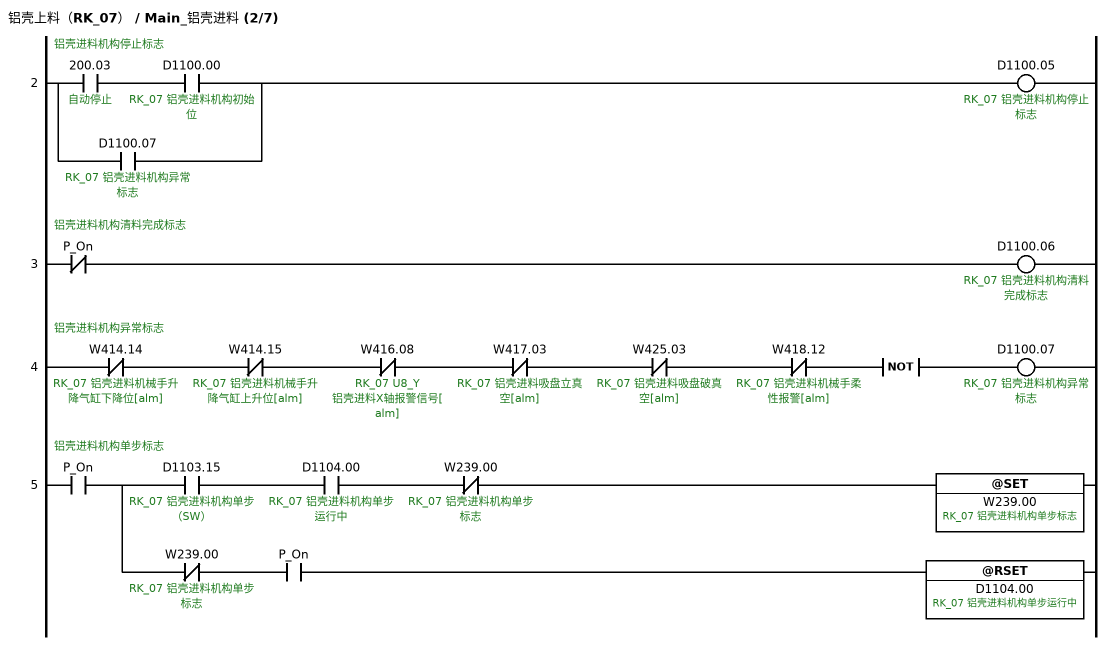
; [picture p552: 铝壳上料（RK_07） / Main_铝壳进料, rungs 2-5]
; rung 2: 铝壳进料机构停止标志
LD 200.03  ; 自动停止
AND D1100.00  ; RK_07 铝壳进料机构初始位
OR D1100.07  ; RK_07 铝壳进料机构异常标志
OUT D1100.05  ; RK_07 铝壳进料机构停止标志
; rung 3: 铝壳进料机构清料完成标志
LDNOT P_On
OUT D1100.06  ; RK_07 铝壳进料机构清料完成标志
; rung 4: 铝壳进料机构异常标志
LDNOT W414.14  ; RK_07 铝壳进料机械手升降气缸下降位[alm]
ANDNOT W414.15  ; RK_07 铝壳进料机械手升降气缸上升位[alm]
ANDNOT W416.08  ; RK_07 U8_Y 铝壳进料X轴报警信号[alm]
ANDNOT W417.03  ; RK_07 铝壳进料吸盘立真空[alm]
ANDNOT W425.03  ; RK_07 铝壳进料吸盘破真空[alm]
ANDNOT W418.12  ; RK_07 铝壳进料机械手柔性报警[alm]
NOT(520)
OUT D1100.07  ; RK_07 铝壳进料机构异常标志
; rung 5: 铝壳进料机构单步标志
LD P_On
OUT TR0
AND D1103.15  ; RK_07 铝壳进料机构单步（SW）
AND D1104.00  ; RK_07 铝壳进料机构单步运行中
ANDNOT W239.00  ; RK_07 铝壳进料机构单步标志
@SET W239.00  ; RK_07 铝壳进料机构单步标志
LD TR0
ANDNOT W239.00  ; RK_07 铝壳进料机构单步标志
AND P_On
@RSET D1104.00  ; RK_07 铝壳进料机构单步运行中

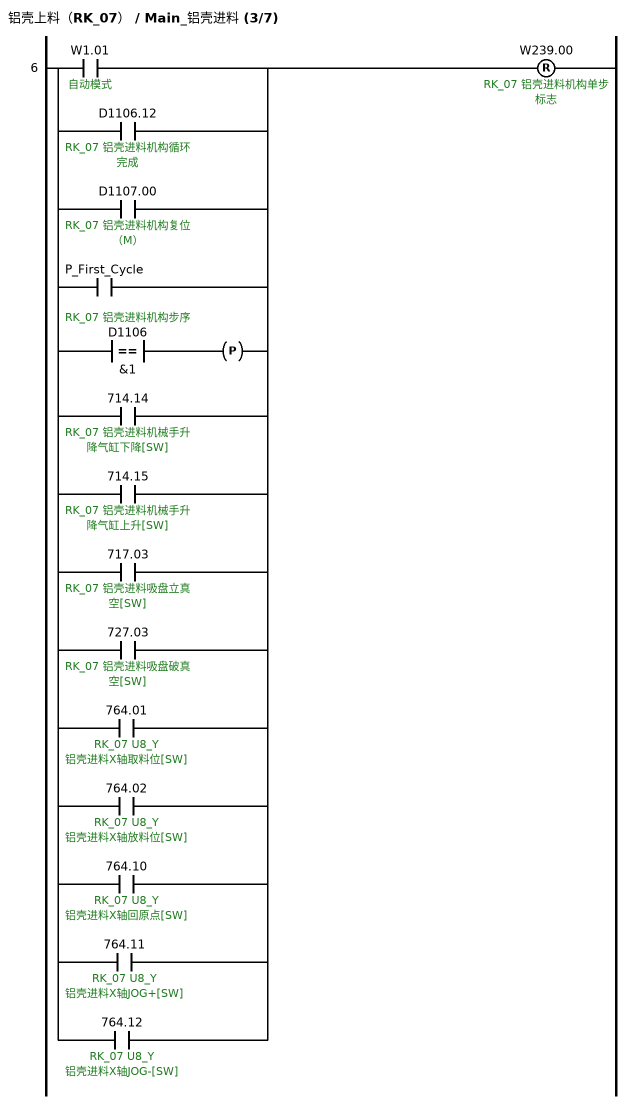
; rung 6
LD W1.01  ; 自动模式
OR D1106.12  ; RK_07 铝壳进料机构循环完成
OR D1107.00  ; RK_07 铝壳进料机构复位（M）
OR P_First_Cycle
LD=(300) D1106 &1  ; RK_07 铝壳进料机构步序
UP(521)
ORLD
OR 714.14  ; RK_07 铝壳进料机械手升降气缸下降[SW]
OR 714.15  ; RK_07 铝壳进料机械手升降气缸上升[SW]
OR 717.03  ; RK_07 铝壳进料吸盘立真空[SW]
OR 727.03  ; RK_07 铝壳进料吸盘破真空[SW]
OR 764.01  ; RK_07 U8_Y 铝壳进料X轴取料位[SW]
OR 764.02  ; RK_07 U8_Y 铝壳进料X轴放料位[SW]
OR 764.10  ; RK_07 U8_Y 铝壳进料X轴回原点[SW]
OR 764.11  ; RK_07 U8_Y 铝壳进料X轴JOG+[SW]
OR 764.12  ; RK_07 U8_Y 铝壳进料X轴JOG-[SW]
RSET W239.00  ; RK_07 铝壳进料机构单步标志

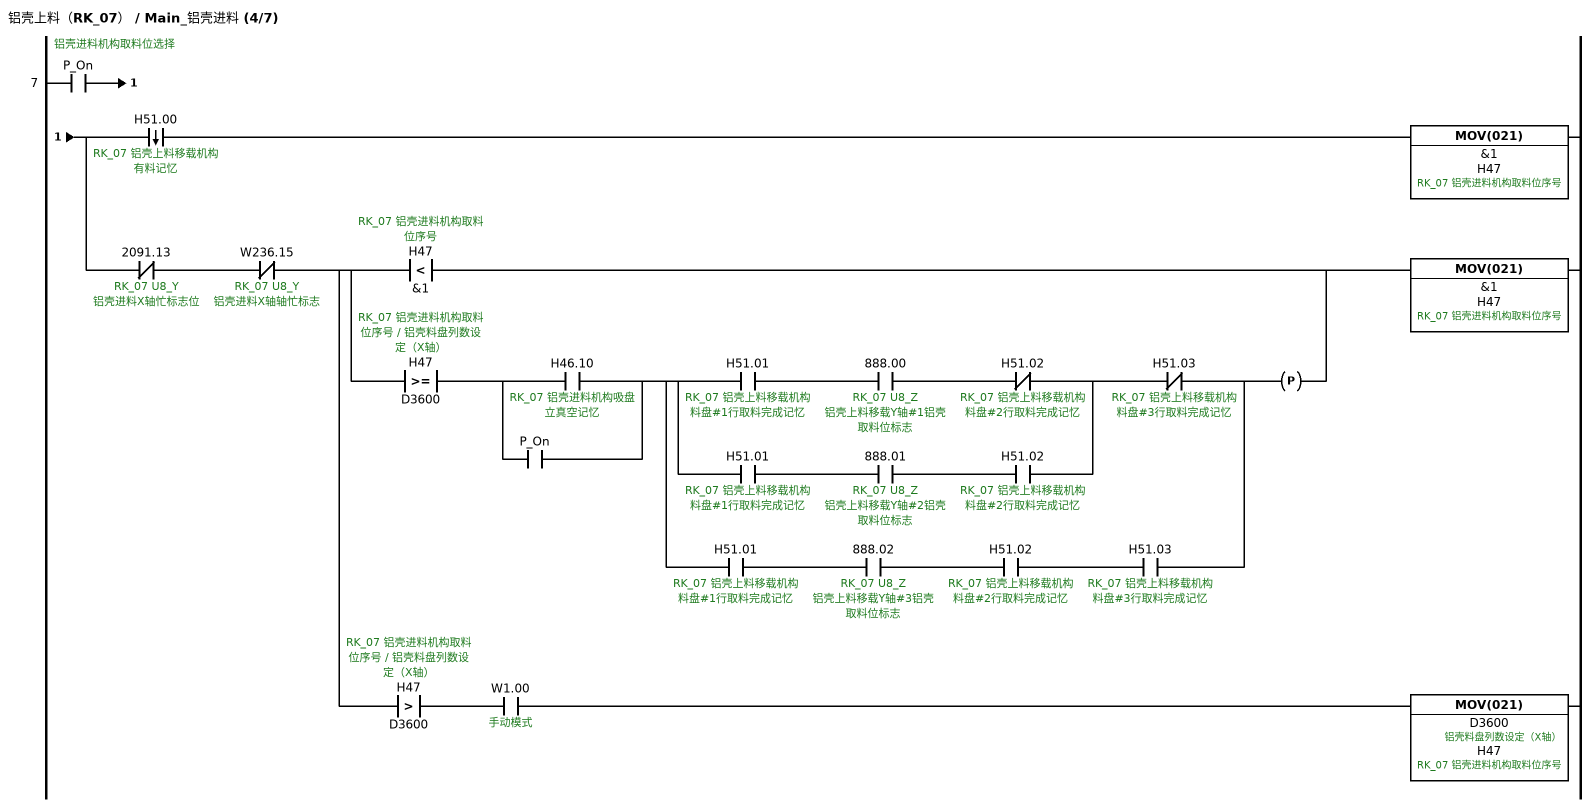
; rung 7: 铝壳进料机构取料位选择
LD P_On
OUT TR0
%AND H51.00  ; RK_07 铝壳上料移载机构有料记忆
MOV(021) &1 H47  ; RK_07 铝壳进料机构取料位序号
LD TR0
ANDNOT 2091.13  ; RK_07 U8_Y 铝壳进料X轴忙标志位
ANDNOT W236.15  ; RK_07 U8_Y 铝壳进料X轴轴忙标志
OUT TR0
LD<(310) H47 &1  ; RK_07 铝壳进料机构取料位序号
LD>=(325) H47 D3600  ; RK_07 铝壳进料机构取料位序号, 铝壳料盘列数设定（X轴）
LD H46.10  ; RK_07 铝壳进料机构吸盘立真空记忆
OR P_On
ANDLD
LD H51.01  ; RK_07 铝壳上料移载机构料盘#1行取料完成记忆
AND 888.00  ; RK_07 U8_Z 铝壳上料移载Y轴#1铝壳取料位标志
ANDNOT H51.02  ; RK_07 铝壳上料移载机构料盘#2行取料完成记忆
LD H51.01  ; RK_07 铝壳上料移载机构料盘#1行取料完成记忆
AND 888.01  ; RK_07 U8_Z 铝壳上料移载Y轴#2铝壳取料位标志
AND H51.02  ; RK_07 铝壳上料移载机构料盘#2行取料完成记忆
ORLD
ANDNOT H51.03  ; RK_07 铝壳上料移载机构料盘#3行取料完成记忆
LD H51.01  ; RK_07 铝壳上料移载机构料盘#1行取料完成记忆
AND 888.02  ; RK_07 U8_Z 铝壳上料移载Y轴#3铝壳取料位标志
AND H51.02  ; RK_07 铝壳上料移载机构料盘#2行取料完成记忆
AND H51.03  ; RK_07 铝壳上料移载机构料盘#3行取料完成记忆
ORLD
ANDLD
UP(521)
ORLD
ANDLD
MOV(021) &1 H47  ; RK_07 铝壳进料机构取料位序号
LD TR0
AND>(320) H47 D3600  ; RK_07 铝壳进料机构取料位序号, 铝壳料盘列数设定（X轴）
AND W1.00  ; 手动模式
MOV(021) D3600 H47  ; 铝壳料盘列数设定（X轴）, RK_07 铝壳进料机构取料位序号

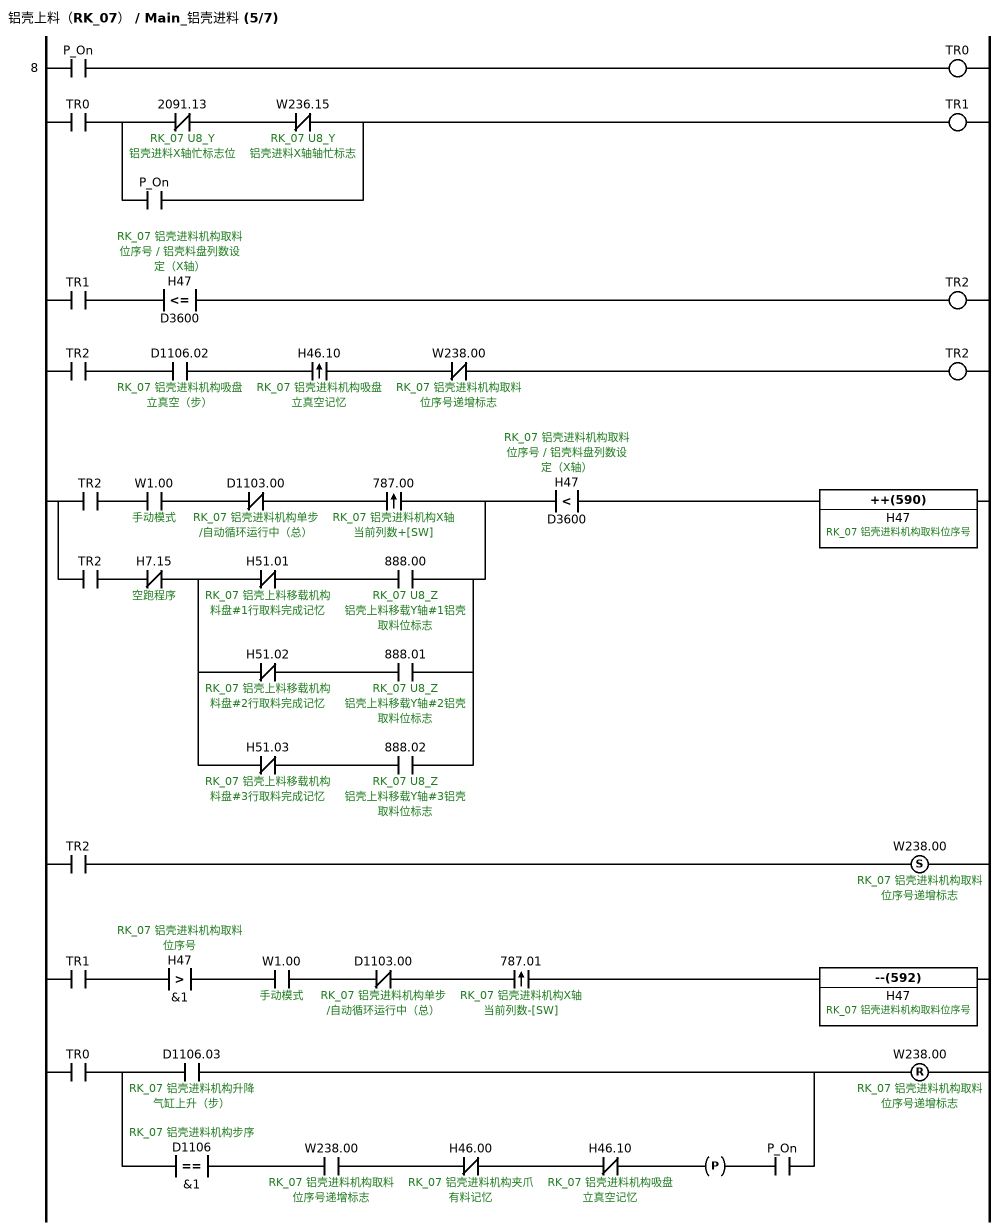
; rung 8
LD P_On
OUT TR0
LDNOT 2091.13  ; RK_07 U8_Y 铝壳进料X轴忙标志位
ANDNOT W236.15  ; RK_07 U8_Y 铝壳进料X轴轴忙标志
OR P_On
ANDLD
OUT TR1
AND<=(315) H47 D3600  ; RK_07 铝壳进料机构取料位序号, 铝壳料盘列数设定（X轴）
OUT TR2
AND W1.00  ; 手动模式
ANDNOT D1103.00  ; RK_07 铝壳进料机构单步/自动循环运行中（总）
@AND 787.00  ; RK_07 铝壳进料机构X轴当前列数+[SW]
LD TR2
AND D1106.02  ; RK_07 铝壳进料机构吸盘立真空（步）
@AND H46.10  ; RK_07 铝壳进料机构吸盘立真空记忆
ANDNOT W238.00  ; RK_07 铝壳进料机构取料位序号递增标志
OUT TR2
ANDNOT H7.15  ; 空跑程序
LDNOT H51.01  ; RK_07 铝壳上料移载机构料盘#1行取料完成记忆
AND 888.00  ; RK_07 U8_Z 铝壳上料移载Y轴#1铝壳取料位标志
LDNOT H51.02  ; RK_07 铝壳上料移载机构料盘#2行取料完成记忆
AND 888.01  ; RK_07 U8_Z 铝壳上料移载Y轴#2铝壳取料位标志
ORLD
LDNOT H51.03  ; RK_07 铝壳上料移载机构料盘#3行取料完成记忆
AND 888.02  ; RK_07 U8_Z 铝壳上料移载Y轴#3铝壳取料位标志
ORLD
ANDLD
ORLD
AND<(310) H47 D3600  ; RK_07 铝壳进料机构取料位序号, 铝壳料盘列数设定（X轴）
++(590) H47  ; RK_07 铝壳进料机构取料位序号
LD TR2
SET W238.00  ; RK_07 铝壳进料机构取料位序号递增标志
LD TR1
AND>(320) H47 &1  ; RK_07 铝壳进料机构取料位序号
AND W1.00  ; 手动模式
ANDNOT D1103.00  ; RK_07 铝壳进料机构单步/自动循环运行中（总）
@AND 787.01  ; RK_07 铝壳进料机构X轴当前列数-[SW]
--(592) H47  ; RK_07 铝壳进料机构取料位序号
LD TR0
LD D1106.03  ; RK_07 铝壳进料机构升降气缸上升（步）
LD=(300) D1106 &1  ; RK_07 铝壳进料机构步序
AND W238.00  ; RK_07 铝壳进料机构取料位序号递增标志
ANDNOT H46.00  ; RK_07 铝壳进料机构夹爪有料记忆
ANDNOT H46.10  ; RK_07 铝壳进料机构吸盘立真空记忆
UP(521)
AND P_On
ORLD
ANDLD
RSET W238.00  ; RK_07 铝壳进料机构取料位序号递增标志

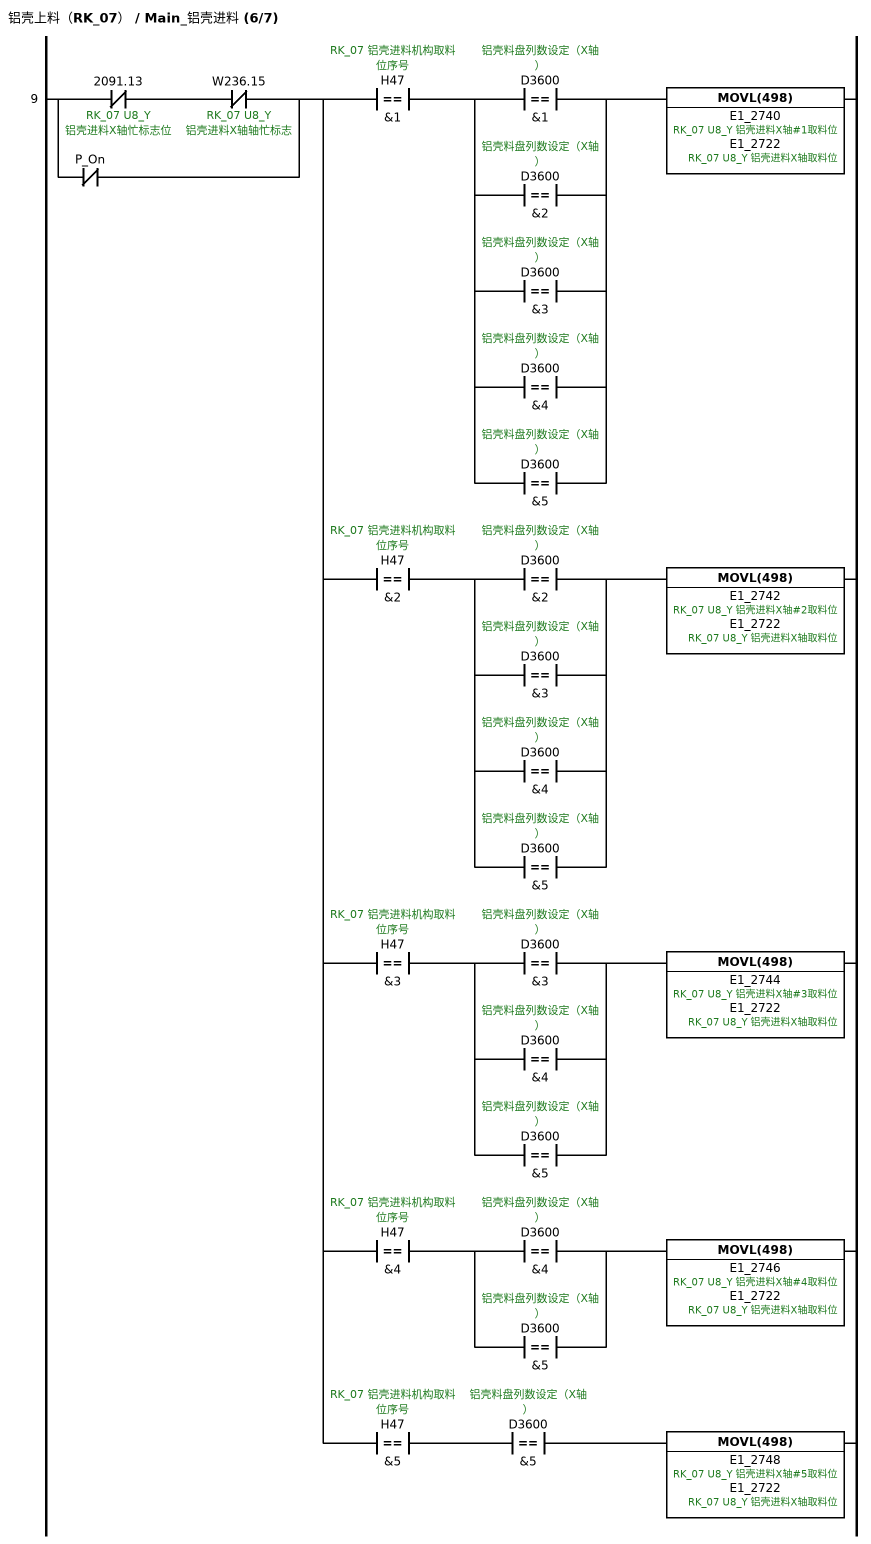
; rung 9
LDNOT 2091.13  ; RK_07 U8_Y 铝壳进料X轴忙标志位
ANDNOT W236.15  ; RK_07 U8_Y 铝壳进料X轴轴忙标志
ORNOT P_On
OUT TR0
AND=(300) H47 &1  ; RK_07 铝壳进料机构取料位序号
LD=(300) D3600 &1  ; 铝壳料盘列数设定（X轴）
OR=(300) D3600 &2  ; 铝壳料盘列数设定（X轴）
OR=(300) D3600 &3  ; 铝壳料盘列数设定（X轴）
OR=(300) D3600 &4  ; 铝壳料盘列数设定（X轴）
OR=(300) D3600 &5  ; 铝壳料盘列数设定（X轴）
ANDLD
MOVL(498) E1_2740 E1_2722  ; RK_07 U8_Y 铝壳进料X轴#1取料位, RK_07 U8_Y 铝壳进料X轴取料位
LD TR0
AND=(300) H47 &2  ; RK_07 铝壳进料机构取料位序号
LD=(300) D3600 &2  ; 铝壳料盘列数设定（X轴）
OR=(300) D3600 &3  ; 铝壳料盘列数设定（X轴）
OR=(300) D3600 &4  ; 铝壳料盘列数设定（X轴）
OR=(300) D3600 &5  ; 铝壳料盘列数设定（X轴）
ANDLD
MOVL(498) E1_2742 E1_2722  ; RK_07 U8_Y 铝壳进料X轴#2取料位, RK_07 U8_Y 铝壳进料X轴取料位
LD TR0
AND=(300) H47 &3  ; RK_07 铝壳进料机构取料位序号
LD=(300) D3600 &3  ; 铝壳料盘列数设定（X轴）
OR=(300) D3600 &4  ; 铝壳料盘列数设定（X轴）
OR=(300) D3600 &5  ; 铝壳料盘列数设定（X轴）
ANDLD
MOVL(498) E1_2744 E1_2722  ; RK_07 U8_Y 铝壳进料X轴#3取料位, RK_07 U8_Y 铝壳进料X轴取料位
LD TR0
AND=(300) H47 &4  ; RK_07 铝壳进料机构取料位序号
LD=(300) D3600 &4  ; 铝壳料盘列数设定（X轴）
OR=(300) D3600 &5  ; 铝壳料盘列数设定（X轴）
ANDLD
MOVL(498) E1_2746 E1_2722  ; RK_07 U8_Y 铝壳进料X轴#4取料位, RK_07 U8_Y 铝壳进料X轴取料位
LD TR0
AND=(300) H47 &5  ; RK_07 铝壳进料机构取料位序号
AND=(300) D3600 &5  ; 铝壳料盘列数设定（X轴）
MOVL(498) E1_2748 E1_2722  ; RK_07 U8_Y 铝壳进料X轴#5取料位, RK_07 U8_Y 铝壳进料X轴取料位

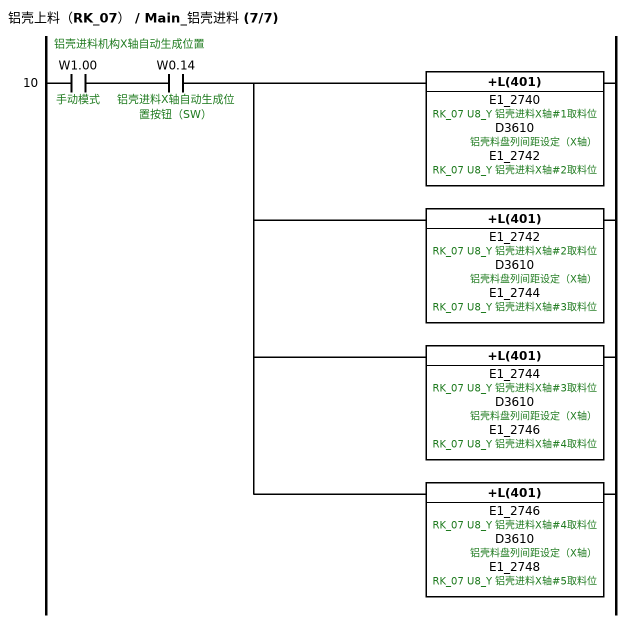
; rung 10: 铝壳进料机构X轴自动生成位置
LD W1.00  ; 手动模式
AND W0.14  ; 铝壳进料X轴自动生成位置按钮（SW）
+L(401) E1_2740 D3610 E1_2742  ; RK_07 U8_Y 铝壳进料X轴#1取料位, 铝壳料盘列间距设定（X轴）, RK_07 U8_Y 铝壳进料X轴#2取料位
+L(401) E1_2742 D3610 E1_2744  ; RK_07 U8_Y 铝壳进料X轴#2取料位, 铝壳料盘列间距设定（X轴）, RK_07 U8_Y 铝壳进料X轴#3取料位
+L(401) E1_2744 D3610 E1_2746  ; RK_07 U8_Y 铝壳进料X轴#3取料位, 铝壳料盘列间距设定（X轴）, RK_07 U8_Y 铝壳进料X轴#4取料位
+L(401) E1_2746 D3610 E1_2748  ; RK_07 U8_Y 铝壳进料X轴#4取料位, 铝壳料盘列间距设定（X轴）, RK_07 U8_Y 铝壳进料X轴#5取料位

### Section Main_铝壳上料移载

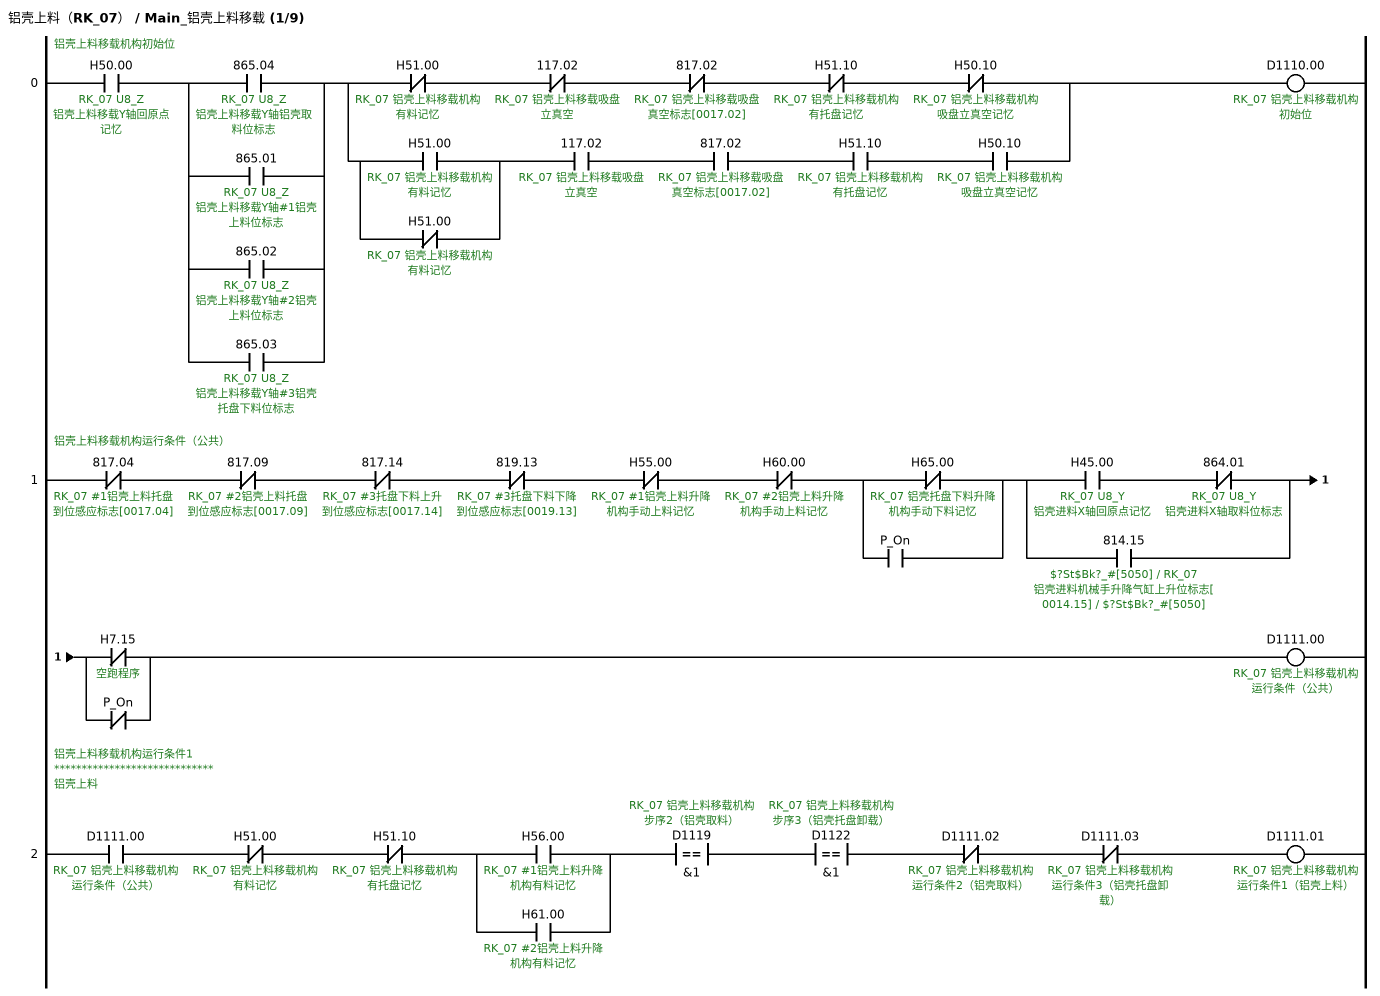
; rung 0: 铝壳上料移载机构初始位
LD H50.00  ; RK_07 U8_Z 铝壳上料移载Y轴回原点记忆
LD 865.04  ; RK_07 U8_Z 铝壳上料移载Y轴铝壳取料位标志
OR 865.01  ; RK_07 U8_Z 铝壳上料移载Y轴#1铝壳上料位标志
OR 865.02  ; RK_07 U8_Z 铝壳上料移载Y轴#2铝壳上料位标志
OR 865.03  ; RK_07 U8_Z 铝壳上料移载Y轴#3铝壳托盘下料位标志
ANDLD
LDNOT H51.00  ; RK_07 铝壳上料移载机构有料记忆
ANDNOT 117.02  ; RK_07 铝壳上料移载吸盘立真空
ANDNOT 817.02  ; RK_07 铝壳上料移载吸盘真空标志[0017.02]
ANDNOT H51.10  ; RK_07 铝壳上料移载机构有托盘记忆
ANDNOT H50.10  ; RK_07 铝壳上料移载机构吸盘立真空记忆
LD H51.00  ; RK_07 铝壳上料移载机构有料记忆
ORNOT H51.00  ; RK_07 铝壳上料移载机构有料记忆
AND 117.02  ; RK_07 铝壳上料移载吸盘立真空
AND 817.02  ; RK_07 铝壳上料移载吸盘真空标志[0017.02]
AND H51.10  ; RK_07 铝壳上料移载机构有托盘记忆
AND H50.10  ; RK_07 铝壳上料移载机构吸盘立真空记忆
ORLD
ANDLD
OUT D1110.00  ; RK_07 铝壳上料移载机构初始位
; rung 1: 铝壳上料移载机构运行条件（公共）
LDNOT 817.04  ; RK_07 #1铝壳上料托盘到位感应标志[0017.04]
ANDNOT 817.09  ; RK_07 #2铝壳上料托盘到位感应标志[0017.09]
ANDNOT 817.14  ; RK_07 #3托盘下料上升到位感应标志[0017.14]
ANDNOT 819.13  ; RK_07 #3托盘下料下降到位感应标志[0019.13]
ANDNOT H55.00  ; RK_07 #1铝壳上料升降机构手动上料记忆
ANDNOT H60.00  ; RK_07 #2铝壳上料升降机构手动上料记忆
LDNOT H65.00  ; RK_07 铝壳托盘下料升降机构手动下料记忆
OR P_On
ANDLD
LD H45.00  ; RK_07 U8_Y 铝壳进料X轴回原点记忆
ANDNOT 864.01  ; RK_07 U8_Y 铝壳进料X轴取料位标志
OR 814.15  ; $?St$Bk?_#[5050] / RK_07 铝壳进料机械手升降气缸上升位标志[0014.15] / $?St$Bk?_#[5050]
ANDLD
LDNOT H7.15  ; 空跑程序
ORNOT P_On
ANDLD
OUT D1111.00  ; RK_07 铝壳上料移载机构运行条件（公共）
; rung 2: 铝壳上料移载机构运行条件1 / ***************************** / 铝壳上料
LD D1111.00  ; RK_07 铝壳上料移载机构运行条件（公共）
ANDNOT H51.00  ; RK_07 铝壳上料移载机构有料记忆
ANDNOT H51.10  ; RK_07 铝壳上料移载机构有托盘记忆
LD H56.00  ; RK_07 #1铝壳上料升降机构有料记忆
OR H61.00  ; RK_07 #2铝壳上料升降机构有料记忆
ANDLD
AND=(300) D1119 &1  ; RK_07 铝壳上料移载机构步序2（铝壳取料）
AND=(300) D1122 &1  ; RK_07 铝壳上料移载机构步序3（铝壳托盘卸载）
ANDNOT D1111.02  ; RK_07 铝壳上料移载机构运行条件2（铝壳取料）
ANDNOT D1111.03  ; RK_07 铝壳上料移载机构运行条件3（铝壳托盘卸载）
OUT D1111.01  ; RK_07 铝壳上料移载机构运行条件1（铝壳上料）

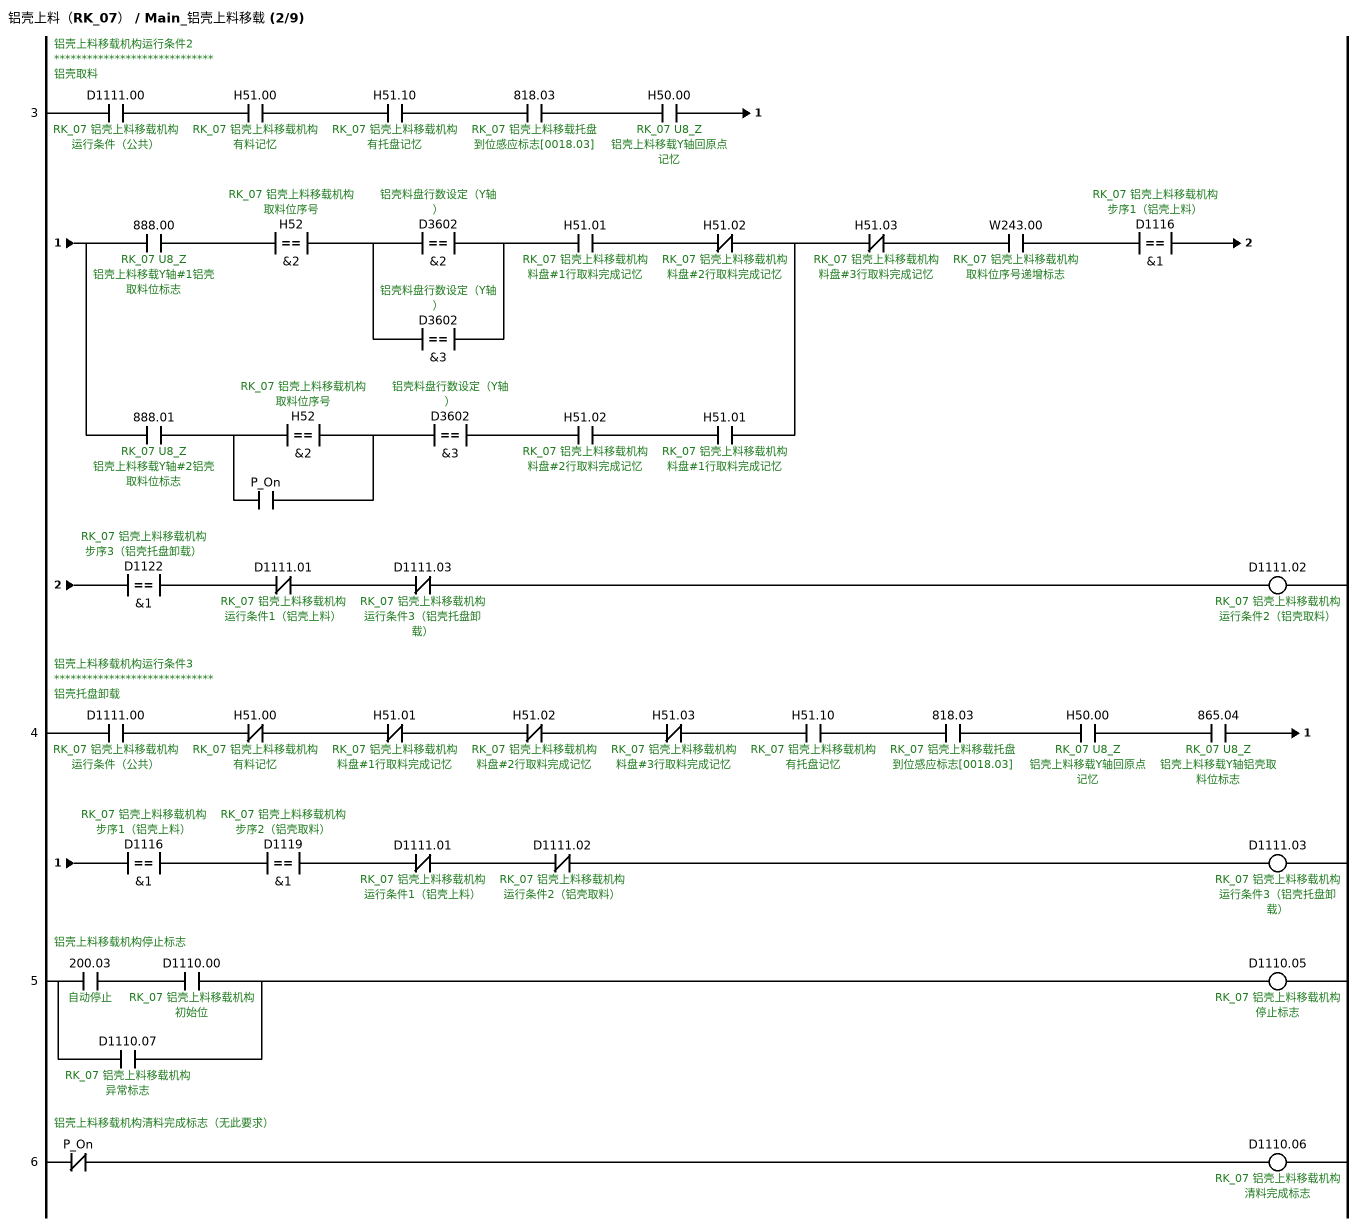
; rung 3: 铝壳上料移载机构运行条件2 / ***************************** / 铝壳取料
LD D1111.00  ; RK_07 铝壳上料移载机构运行条件（公共）
AND H51.00  ; RK_07 铝壳上料移载机构有料记忆
AND H51.10  ; RK_07 铝壳上料移载机构有托盘记忆
AND 818.03  ; RK_07 铝壳上料移载托盘到位感应标志[0018.03]
AND H50.00  ; RK_07 U8_Z 铝壳上料移载Y轴回原点记忆
LD 888.00  ; RK_07 U8_Z 铝壳上料移载Y轴#1铝壳取料位标志
AND=(300) H52 &2  ; RK_07 铝壳上料移载机构取料位序号
LD=(300) D3602 &2  ; 铝壳料盘行数设定（Y轴）
OR=(300) D3602 &3  ; 铝壳料盘行数设定（Y轴）
ANDLD
AND H51.01  ; RK_07 铝壳上料移载机构料盘#1行取料完成记忆
ANDNOT H51.02  ; RK_07 铝壳上料移载机构料盘#2行取料完成记忆
LD 888.01  ; RK_07 U8_Z 铝壳上料移载Y轴#2铝壳取料位标志
LD=(300) H52 &2  ; RK_07 铝壳上料移载机构取料位序号
OR P_On
ANDLD
AND=(300) D3602 &3  ; 铝壳料盘行数设定（Y轴）
AND H51.02  ; RK_07 铝壳上料移载机构料盘#2行取料完成记忆
AND H51.01  ; RK_07 铝壳上料移载机构料盘#1行取料完成记忆
ORLD
ANDLD
ANDNOT H51.03  ; RK_07 铝壳上料移载机构料盘#3行取料完成记忆
AND W243.00  ; RK_07 铝壳上料移载机构取料位序号递增标志
AND=(300) D1116 &1  ; RK_07 铝壳上料移载机构步序1（铝壳上料）
AND=(300) D1122 &1  ; RK_07 铝壳上料移载机构步序3（铝壳托盘卸载）
ANDNOT D1111.01  ; RK_07 铝壳上料移载机构运行条件1（铝壳上料）
ANDNOT D1111.03  ; RK_07 铝壳上料移载机构运行条件3（铝壳托盘卸载）
OUT D1111.02  ; RK_07 铝壳上料移载机构运行条件2（铝壳取料）
; rung 4: 铝壳上料移载机构运行条件3 / ***************************** / 铝壳托盘卸载
LD D1111.00  ; RK_07 铝壳上料移载机构运行条件（公共）
ANDNOT H51.00  ; RK_07 铝壳上料移载机构有料记忆
ANDNOT H51.01  ; RK_07 铝壳上料移载机构料盘#1行取料完成记忆
ANDNOT H51.02  ; RK_07 铝壳上料移载机构料盘#2行取料完成记忆
ANDNOT H51.03  ; RK_07 铝壳上料移载机构料盘#3行取料完成记忆
AND H51.10  ; RK_07 铝壳上料移载机构有托盘记忆
AND 818.03  ; RK_07 铝壳上料移载托盘到位感应标志[0018.03]
AND H50.00  ; RK_07 U8_Z 铝壳上料移载Y轴回原点记忆
AND 865.04  ; RK_07 U8_Z 铝壳上料移载Y轴铝壳取料位标志
AND=(300) D1116 &1  ; RK_07 铝壳上料移载机构步序1（铝壳上料）
AND=(300) D1119 &1  ; RK_07 铝壳上料移载机构步序2（铝壳取料）
ANDNOT D1111.01  ; RK_07 铝壳上料移载机构运行条件1（铝壳上料）
ANDNOT D1111.02  ; RK_07 铝壳上料移载机构运行条件2（铝壳取料）
OUT D1111.03  ; RK_07 铝壳上料移载机构运行条件3（铝壳托盘卸载）
; rung 5: 铝壳上料移载机构停止标志
LD 200.03  ; 自动停止
AND D1110.00  ; RK_07 铝壳上料移载机构初始位
OR D1110.07  ; RK_07 铝壳上料移载机构异常标志
OUT D1110.05  ; RK_07 铝壳上料移载机构停止标志
; rung 6: 铝壳上料移载机构清料完成标志（无此要求）
LDNOT P_On
OUT D1110.06  ; RK_07 铝壳上料移载机构清料完成标志

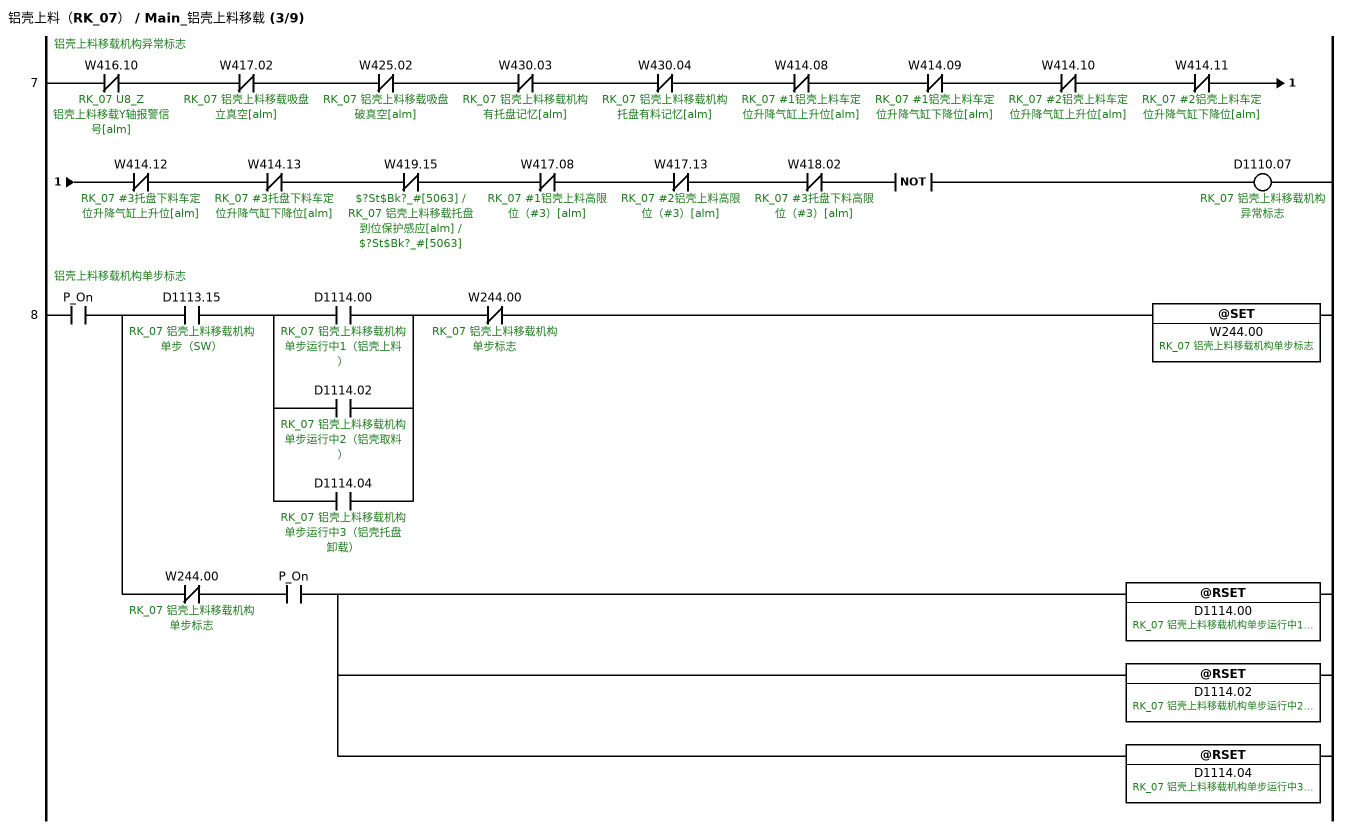
; rung 7: 铝壳上料移载机构异常标志
LDNOT W416.10  ; RK_07 U8_Z 铝壳上料移载Y轴报警信号[alm]
ANDNOT W417.02  ; RK_07 铝壳上料移载吸盘立真空[alm]
ANDNOT W425.02  ; RK_07 铝壳上料移载吸盘破真空[alm]
ANDNOT W430.03  ; RK_07 铝壳上料移载机构有托盘记忆[alm]
ANDNOT W430.04  ; RK_07 铝壳上料移载机构托盘有料记忆[alm]
ANDNOT W414.08  ; RK_07 #1铝壳上料车定位升降气缸上升位[alm]
ANDNOT W414.09  ; RK_07 #1铝壳上料车定位升降气缸下降位[alm]
ANDNOT W414.10  ; RK_07 #2铝壳上料车定位升降气缸上升位[alm]
ANDNOT W414.11  ; RK_07 #2铝壳上料车定位升降气缸下降位[alm]
ANDNOT W414.12  ; RK_07 #3托盘下料车定位升降气缸上升位[alm]
ANDNOT W414.13  ; RK_07 #3托盘下料车定位升降气缸下降位[alm]
ANDNOT W419.15  ; $?St$Bk?_#[5063] / RK_07 铝壳上料移载托盘到位保护感应[alm] / $?St$Bk?_#[5063]
ANDNOT W417.08  ; RK_07 #1铝壳上料高限位（#3）[alm]
ANDNOT W417.13  ; RK_07 #2铝壳上料高限位（#3）[alm]
ANDNOT W418.02  ; RK_07 #3托盘下料高限位（#3）[alm]
NOT(520)
OUT D1110.07  ; RK_07 铝壳上料移载机构异常标志
; rung 8: 铝壳上料移载机构单步标志
LD P_On
OUT TR0
AND D1113.15  ; RK_07 铝壳上料移载机构单步（SW）
LD D1114.00  ; RK_07 铝壳上料移载机构单步运行中1（铝壳上料）
OR D1114.02  ; RK_07 铝壳上料移载机构单步运行中2（铝壳取料）
OR D1114.04  ; RK_07 铝壳上料移载机构单步运行中3（铝壳托盘卸载）
ANDLD
ANDNOT W244.00  ; RK_07 铝壳上料移载机构单步标志
@SET W244.00  ; RK_07 铝壳上料移载机构单步标志
LD TR0
ANDNOT W244.00  ; RK_07 铝壳上料移载机构单步标志
AND P_On
@RSET D1114.00  ; RK_07 铝壳上料移载机构单步运行中1（铝壳上料）
@RSET D1114.02  ; RK_07 铝壳上料移载机构单步运行中2（铝壳取料）
@RSET D1114.04  ; RK_07 铝壳上料移载机构单步运行中3（铝壳托盘卸载）

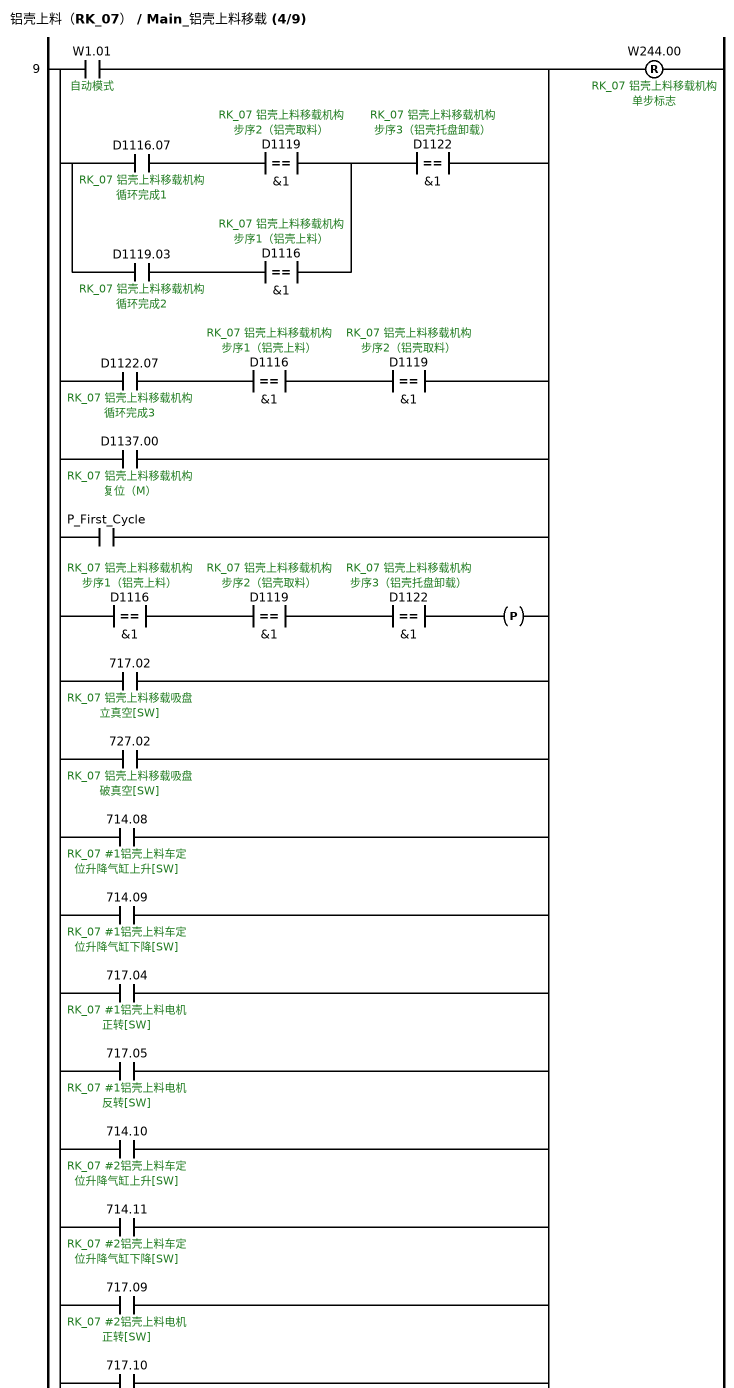

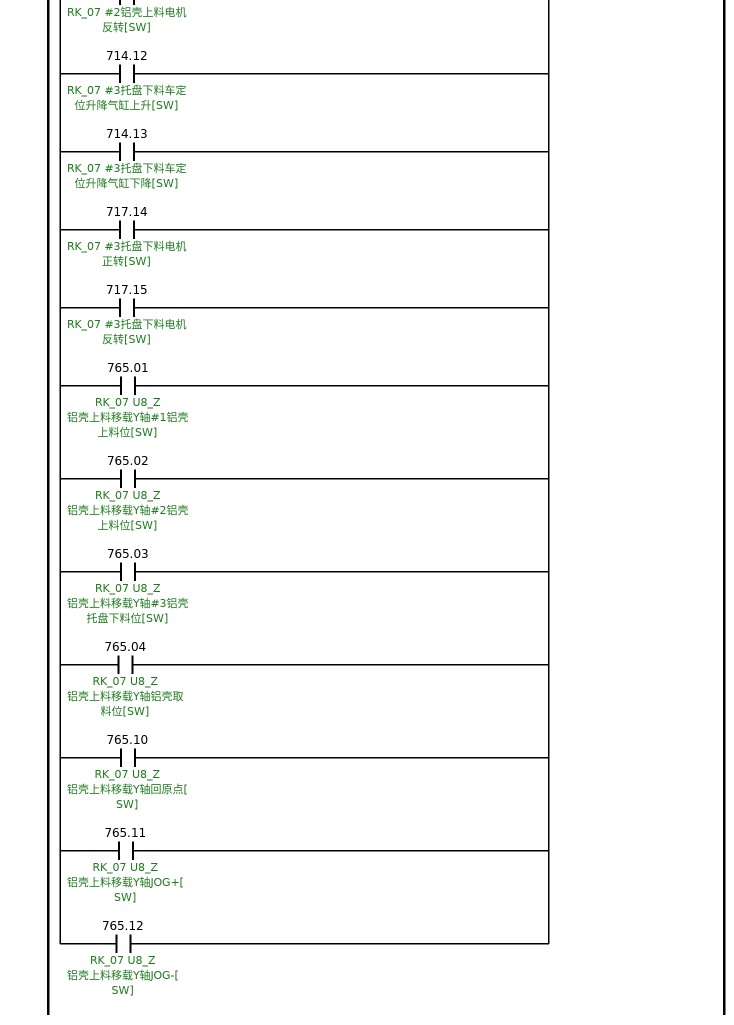
; rung 9
LD W1.01  ; 自动模式
LD D1116.07  ; RK_07 铝壳上料移载机构循环完成1
AND=(300) D1119 &1  ; RK_07 铝壳上料移载机构步序2（铝壳取料）
LD D1119.03  ; RK_07 铝壳上料移载机构循环完成2
AND=(300) D1116 &1  ; RK_07 铝壳上料移载机构步序1（铝壳上料）
ORLD
AND=(300) D1122 &1  ; RK_07 铝壳上料移载机构步序3（铝壳托盘卸载）
ORLD
LD D1122.07  ; RK_07 铝壳上料移载机构循环完成3
AND=(300) D1116 &1  ; RK_07 铝壳上料移载机构步序1（铝壳上料）
AND=(300) D1119 &1  ; RK_07 铝壳上料移载机构步序2（铝壳取料）
ORLD
OR D1137.00  ; RK_07 铝壳上料移载机构复位（M）
OR P_First_Cycle
LD=(300) D1116 &1  ; RK_07 铝壳上料移载机构步序1（铝壳上料）
AND=(300) D1119 &1  ; RK_07 铝壳上料移载机构步序2（铝壳取料）
AND=(300) D1122 &1  ; RK_07 铝壳上料移载机构步序3（铝壳托盘卸载）
UP(521)
ORLD
LD 717.02  ; RK_07 铝壳上料移载吸盘立真空[SW]
OR 727.02  ; RK_07 铝壳上料移载吸盘破真空[SW]
OR 714.08  ; RK_07 #1铝壳上料车定位升降气缸上升[SW]
OR 714.09  ; RK_07 #1铝壳上料车定位升降气缸下降[SW]
OR 717.04  ; RK_07 #1铝壳上料电机正转[SW]
OR 717.05  ; RK_07 #1铝壳上料电机反转[SW]
OR 714.10  ; RK_07 #2铝壳上料车定位升降气缸上升[SW]
OR 714.11  ; RK_07 #2铝壳上料车定位升降气缸下降[SW]
OR 717.09  ; RK_07 #2铝壳上料电机正转[SW]
OR 717.10  ; RK_07 #2铝壳上料电机反转[SW]
OR 714.12  ; RK_07 #3托盘下料车定位升降气缸上升[SW]
OR 714.13  ; RK_07 #3托盘下料车定位升降气缸下降[SW]
OR 717.14  ; RK_07 #3托盘下料电机正转[SW]
OR 717.15  ; RK_07 #3托盘下料电机反转[SW]
OR 765.01  ; RK_07 U8_Z 铝壳上料移载Y轴#1铝壳上料位[SW]
OR 765.02  ; RK_07 U8_Z 铝壳上料移载Y轴#2铝壳上料位[SW]
OR 765.03  ; RK_07 U8_Z 铝壳上料移载Y轴#3铝壳托盘下料位[SW]
OR 765.04  ; RK_07 U8_Z 铝壳上料移载Y轴铝壳取料位[SW]
OR 765.10  ; RK_07 U8_Z 铝壳上料移载Y轴回原点[SW]
OR 765.11  ; RK_07 U8_Z 铝壳上料移载Y轴JOG+[SW]
OR 765.12  ; RK_07 U8_Z 铝壳上料移载Y轴JOG-[SW]
ORLD
RSET W244.00  ; RK_07 铝壳上料移载机构单步标志

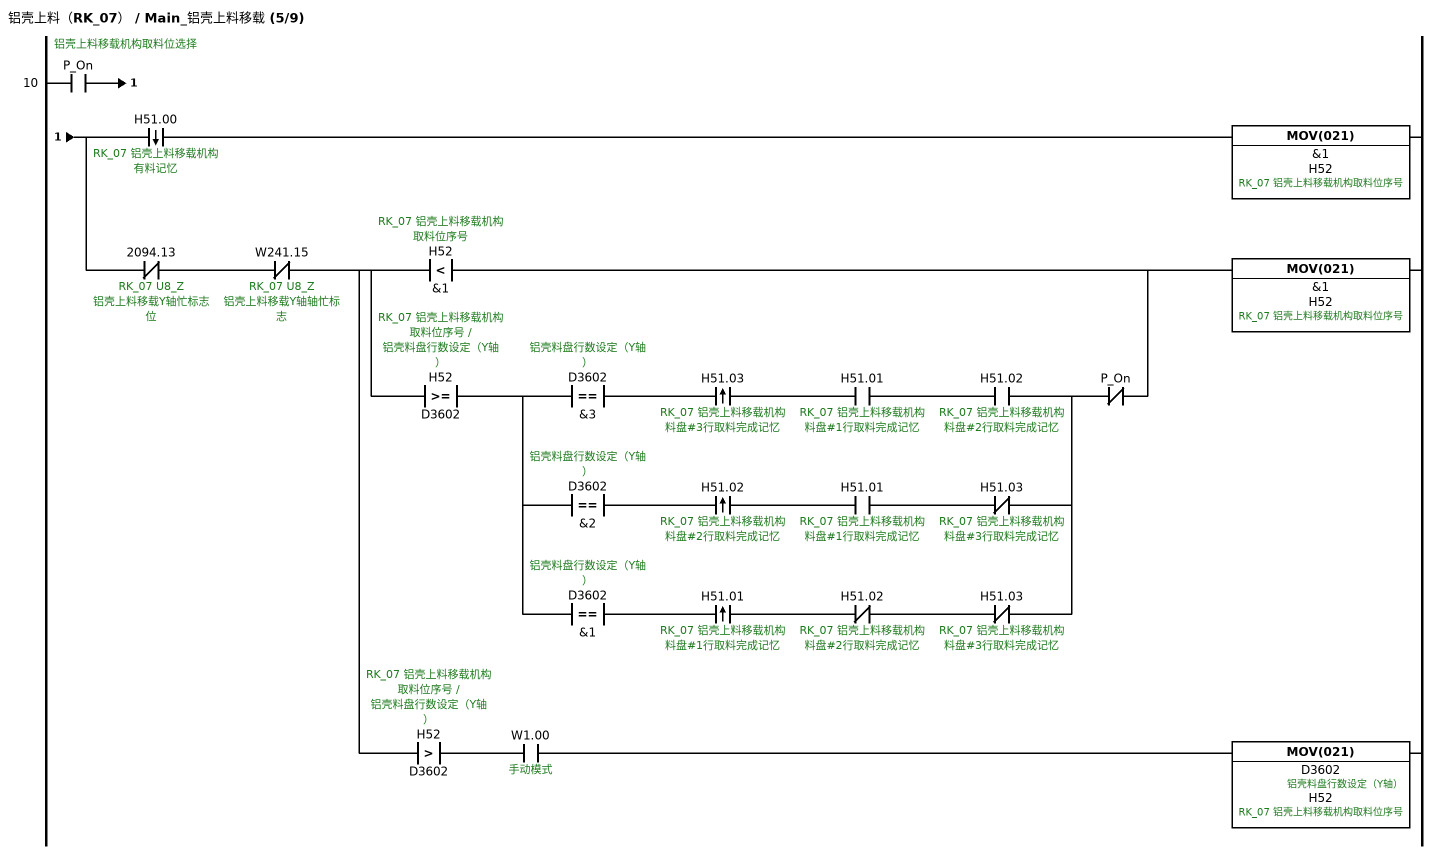
; rung 10: 铝壳上料移载机构取料位选择
LD P_On
OUT TR0
%AND H51.00  ; RK_07 铝壳上料移载机构有料记忆
MOV(021) &1 H52  ; RK_07 铝壳上料移载机构取料位序号
LD TR0
ANDNOT 2094.13  ; RK_07 U8_Z 铝壳上料移载Y轴忙标志位
ANDNOT W241.15  ; RK_07 U8_Z 铝壳上料移载Y轴轴忙标志
OUT TR0
LD<(310) H52 &1  ; RK_07 铝壳上料移载机构取料位序号
LD>=(325) H52 D3602  ; RK_07 铝壳上料移载机构取料位序号, 铝壳料盘行数设定（Y轴）
LD=(300) D3602 &3  ; 铝壳料盘行数设定（Y轴）
@AND H51.03  ; RK_07 铝壳上料移载机构料盘#3行取料完成记忆
AND H51.01  ; RK_07 铝壳上料移载机构料盘#1行取料完成记忆
AND H51.02  ; RK_07 铝壳上料移载机构料盘#2行取料完成记忆
LD=(300) D3602 &2  ; 铝壳料盘行数设定（Y轴）
@AND H51.02  ; RK_07 铝壳上料移载机构料盘#2行取料完成记忆
AND H51.01  ; RK_07 铝壳上料移载机构料盘#1行取料完成记忆
ANDNOT H51.03  ; RK_07 铝壳上料移载机构料盘#3行取料完成记忆
ORLD
LD=(300) D3602 &1  ; 铝壳料盘行数设定（Y轴）
@AND H51.01  ; RK_07 铝壳上料移载机构料盘#1行取料完成记忆
ANDNOT H51.02  ; RK_07 铝壳上料移载机构料盘#2行取料完成记忆
ANDNOT H51.03  ; RK_07 铝壳上料移载机构料盘#3行取料完成记忆
ORLD
ANDLD
ANDNOT P_On
ORLD
ANDLD
MOV(021) &1 H52  ; RK_07 铝壳上料移载机构取料位序号
LD TR0
AND>(320) H52 D3602  ; RK_07 铝壳上料移载机构取料位序号, 铝壳料盘行数设定（Y轴）
AND W1.00  ; 手动模式
MOV(021) D3602 H52  ; 铝壳料盘行数设定（Y轴）, RK_07 铝壳上料移载机构取料位序号

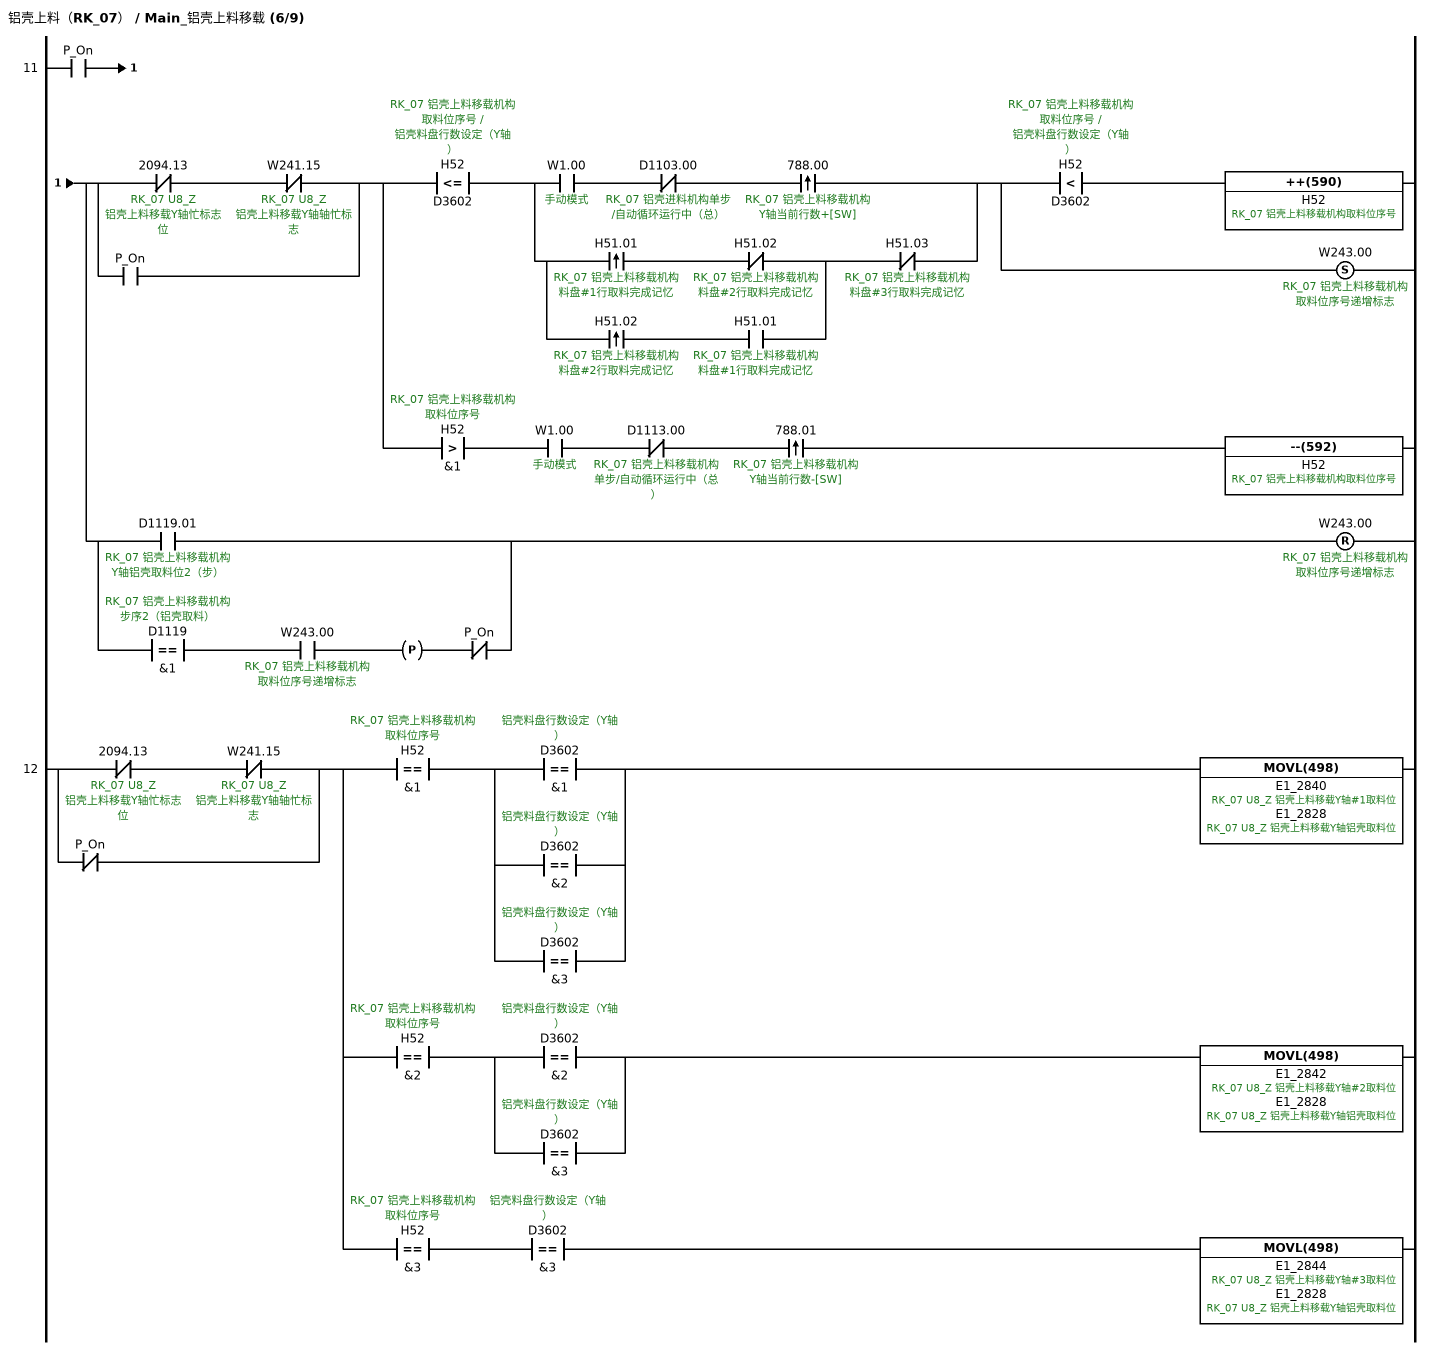
; rung 11
LD P_On
OUT TR0
LDNOT 2094.13  ; RK_07 U8_Z 铝壳上料移载Y轴忙标志位
ANDNOT W241.15  ; RK_07 U8_Z 铝壳上料移载Y轴轴忙标志
OR P_On
ANDLD
OUT TR1
AND<=(315) H52 D3602  ; RK_07 铝壳上料移载机构取料位序号, 铝壳料盘行数设定（Y轴）
LD W1.00  ; 手动模式
ANDNOT D1103.00  ; RK_07 铝壳进料机构单步/自动循环运行中（总）
@AND 788.00  ; RK_07 铝壳上料移载机构Y轴当前行数+[SW]
@LD H51.01  ; RK_07 铝壳上料移载机构料盘#1行取料完成记忆
ANDNOT H51.02  ; RK_07 铝壳上料移载机构料盘#2行取料完成记忆
@LD H51.02  ; RK_07 铝壳上料移载机构料盘#2行取料完成记忆
AND H51.01  ; RK_07 铝壳上料移载机构料盘#1行取料完成记忆
ORLD
ANDNOT H51.03  ; RK_07 铝壳上料移载机构料盘#3行取料完成记忆
ORLD
ANDLD
OUT TR2
AND<(310) H52 D3602  ; RK_07 铝壳上料移载机构取料位序号, 铝壳料盘行数设定（Y轴）
++(590) H52  ; RK_07 铝壳上料移载机构取料位序号
LD TR2
SET W243.00  ; RK_07 铝壳上料移载机构取料位序号递增标志
LD TR1
AND>(320) H52 &1  ; RK_07 铝壳上料移载机构取料位序号
AND W1.00  ; 手动模式
ANDNOT D1113.00  ; RK_07 铝壳上料移载机构单步/自动循环运行中（总）
@AND 788.01  ; RK_07 铝壳上料移载机构Y轴当前行数-[SW]
--(592) H52  ; RK_07 铝壳上料移载机构取料位序号
LD TR0
LD D1119.01  ; RK_07 铝壳上料移载机构Y轴铝壳取料位2（步）
LD=(300) D1119 &1  ; RK_07 铝壳上料移载机构步序2（铝壳取料）
AND W243.00  ; RK_07 铝壳上料移载机构取料位序号递增标志
UP(521)
ANDNOT P_On
ORLD
ANDLD
RSET W243.00  ; RK_07 铝壳上料移载机构取料位序号递增标志
; rung 12
LDNOT 2094.13  ; RK_07 U8_Z 铝壳上料移载Y轴忙标志位
ANDNOT W241.15  ; RK_07 U8_Z 铝壳上料移载Y轴轴忙标志
ORNOT P_On
OUT TR0
AND=(300) H52 &1  ; RK_07 铝壳上料移载机构取料位序号
LD=(300) D3602 &1  ; 铝壳料盘行数设定（Y轴）
OR=(300) D3602 &2  ; 铝壳料盘行数设定（Y轴）
OR=(300) D3602 &3  ; 铝壳料盘行数设定（Y轴）
ANDLD
MOVL(498) E1_2840 E1_2828  ; RK_07 U8_Z 铝壳上料移载Y轴#1取料位, RK_07 U8_Z 铝壳上料移载Y轴铝壳取料位
LD TR0
AND=(300) H52 &2  ; RK_07 铝壳上料移载机构取料位序号
LD=(300) D3602 &2  ; 铝壳料盘行数设定（Y轴）
OR=(300) D3602 &3  ; 铝壳料盘行数设定（Y轴）
ANDLD
MOVL(498) E1_2842 E1_2828  ; RK_07 U8_Z 铝壳上料移载Y轴#2取料位, RK_07 U8_Z 铝壳上料移载Y轴铝壳取料位
LD TR0
AND=(300) H52 &3  ; RK_07 铝壳上料移载机构取料位序号
AND=(300) D3602 &3  ; 铝壳料盘行数设定（Y轴）
MOVL(498) E1_2844 E1_2828  ; RK_07 U8_Z 铝壳上料移载Y轴#3取料位, RK_07 U8_Z 铝壳上料移载Y轴铝壳取料位

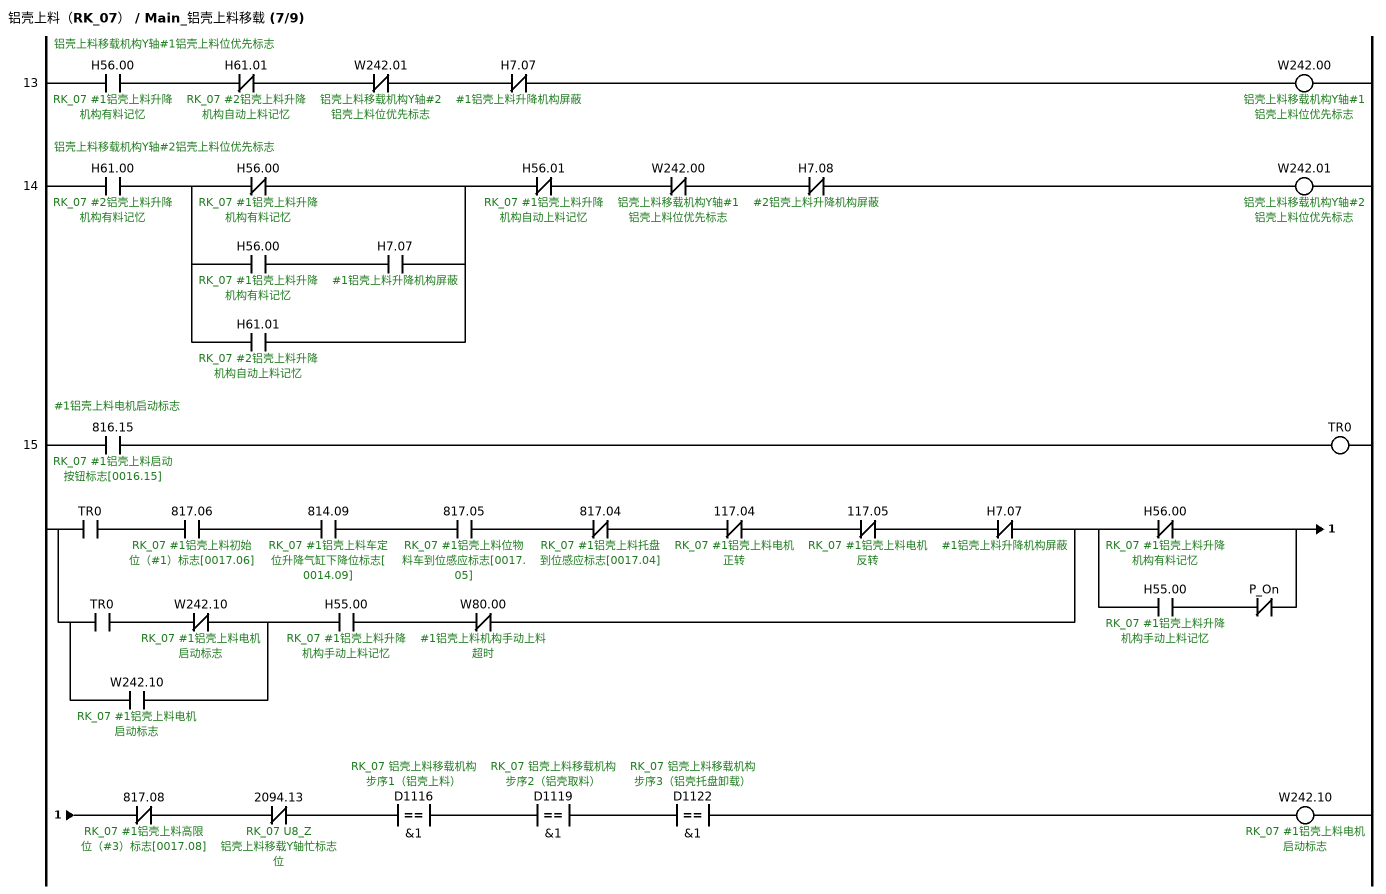
; rung 13: 铝壳上料移载机构Y轴#1铝壳上料位优先标志
LD H56.00  ; RK_07 #1铝壳上料升降机构有料记忆
ANDNOT H61.01  ; RK_07 #2铝壳上料升降机构自动上料记忆
ANDNOT W242.01  ; 铝壳上料移载机构Y轴#2铝壳上料位优先标志
ANDNOT H7.07  ; #1铝壳上料升降机构屏蔽
OUT W242.00  ; 铝壳上料移载机构Y轴#1铝壳上料位优先标志
; rung 14: 铝壳上料移载机构Y轴#2铝壳上料位优先标志
LD H61.00  ; RK_07 #2铝壳上料升降机构有料记忆
LDNOT H56.00  ; RK_07 #1铝壳上料升降机构有料记忆
LD H56.00  ; RK_07 #1铝壳上料升降机构有料记忆
AND H7.07  ; #1铝壳上料升降机构屏蔽
ORLD
OR H61.01  ; RK_07 #2铝壳上料升降机构自动上料记忆
ANDLD
ANDNOT H56.01  ; RK_07 #1铝壳上料升降机构自动上料记忆
ANDNOT W242.00  ; 铝壳上料移载机构Y轴#1铝壳上料位优先标志
ANDNOT H7.08  ; #2铝壳上料升降机构屏蔽
OUT W242.01  ; 铝壳上料移载机构Y轴#2铝壳上料位优先标志
; rung 15: #1铝壳上料电机启动标志
LD 816.15  ; RK_07 #1铝壳上料启动按钮标志[0016.15]
OUT TR0
AND 817.06  ; RK_07 #1铝壳上料初始位（#1）标志[0017.06]
AND 814.09  ; RK_07 #1铝壳上料车定位升降气缸下降位标志[0014.09]
AND 817.05  ; RK_07 #1铝壳上料位物料车到位感应标志[0017.05]
ANDNOT 817.04  ; RK_07 #1铝壳上料托盘到位感应标志[0017.04]
ANDNOT 117.04  ; RK_07 #1铝壳上料电机正转
ANDNOT 117.05  ; RK_07 #1铝壳上料电机反转
ANDNOT H7.07  ; #1铝壳上料升降机构屏蔽
LD TR0
ANDNOT W242.10  ; RK_07 #1铝壳上料电机启动标志
OR W242.10  ; RK_07 #1铝壳上料电机启动标志
AND H55.00  ; RK_07 #1铝壳上料升降机构手动上料记忆
ANDNOT W80.00  ; #1铝壳上料机构手动上料超时
ORLD
LDNOT H56.00  ; RK_07 #1铝壳上料升降机构有料记忆
LD H55.00  ; RK_07 #1铝壳上料升降机构手动上料记忆
ANDNOT P_On
ORLD
ANDLD
ANDNOT 817.08  ; RK_07 #1铝壳上料高限位（#3）标志[0017.08]
ANDNOT 2094.13  ; RK_07 U8_Z 铝壳上料移载Y轴忙标志位
AND=(300) D1116 &1  ; RK_07 铝壳上料移载机构步序1（铝壳上料）
AND=(300) D1119 &1  ; RK_07 铝壳上料移载机构步序2（铝壳取料）
AND=(300) D1122 &1  ; RK_07 铝壳上料移载机构步序3（铝壳托盘卸载）
OUT W242.10  ; RK_07 #1铝壳上料电机启动标志

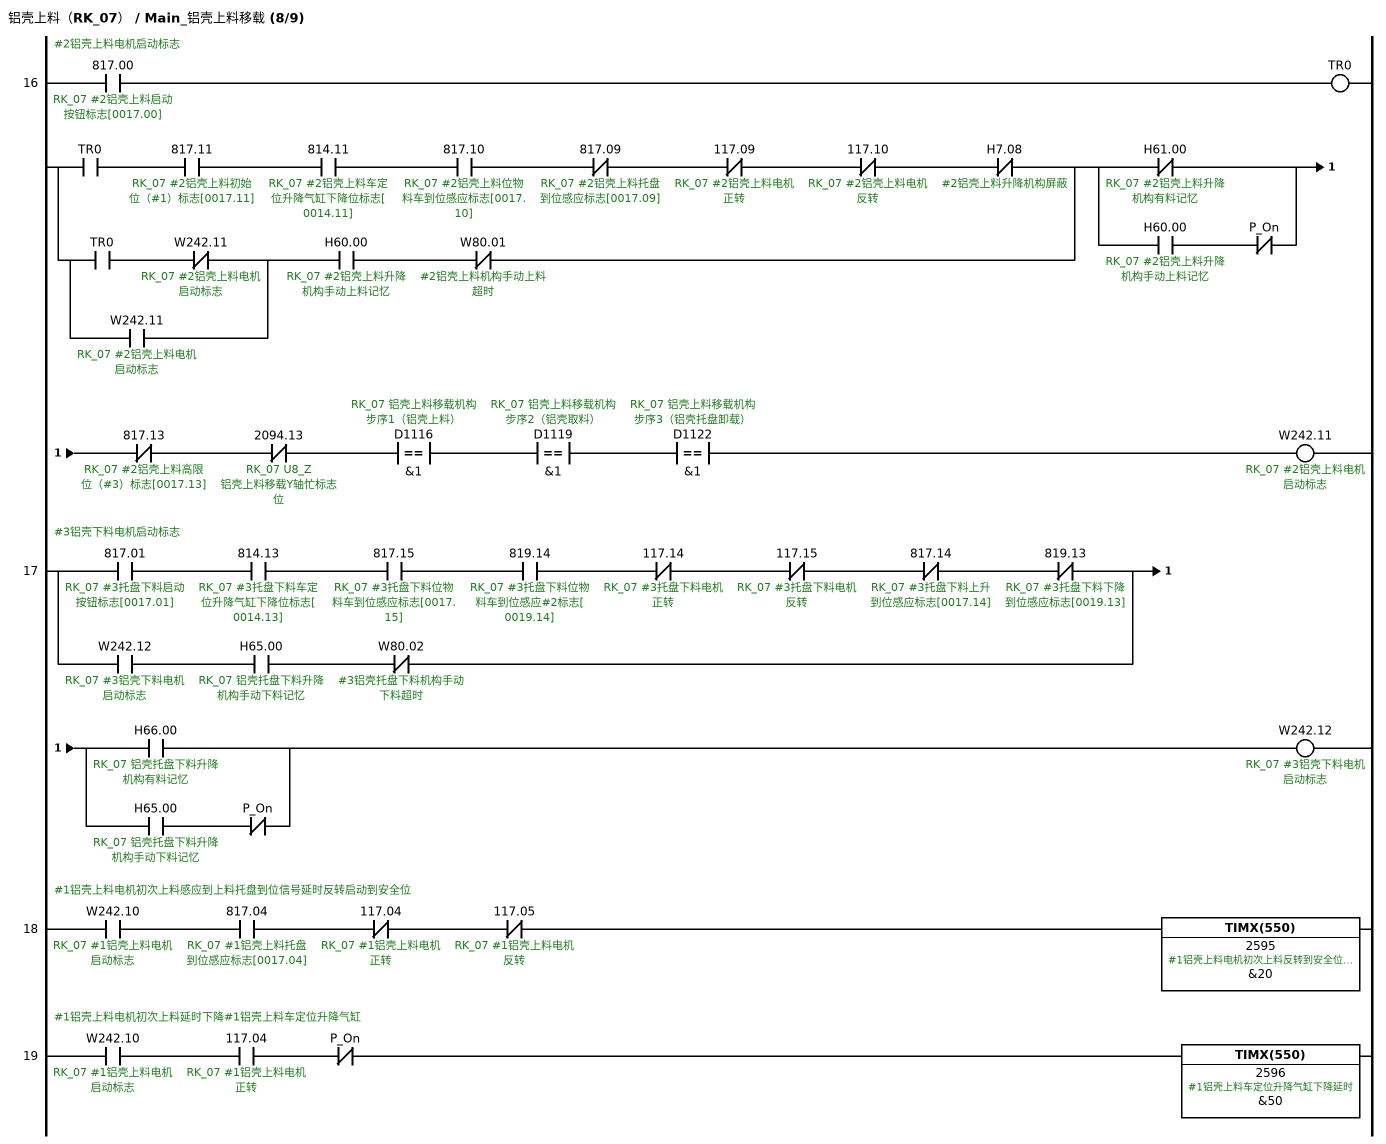
; rung 16: #2铝壳上料电机启动标志
LD 817.00  ; RK_07 #2铝壳上料启动按钮标志[0017.00]
OUT TR0
AND 817.11  ; RK_07 #2铝壳上料初始位（#1）标志[0017.11]
AND 814.11  ; RK_07 #2铝壳上料车定位升降气缸下降位标志[0014.11]
AND 817.10  ; RK_07 #2铝壳上料位物料车到位感应标志[0017.10]
ANDNOT 817.09  ; RK_07 #2铝壳上料托盘到位感应标志[0017.09]
ANDNOT 117.09  ; RK_07 #2铝壳上料电机正转
ANDNOT 117.10  ; RK_07 #2铝壳上料电机反转
ANDNOT H7.08  ; #2铝壳上料升降机构屏蔽
LD TR0
ANDNOT W242.11  ; RK_07 #2铝壳上料电机启动标志
OR W242.11  ; RK_07 #2铝壳上料电机启动标志
AND H60.00  ; RK_07 #2铝壳上料升降机构手动上料记忆
ANDNOT W80.01  ; #2铝壳上料机构手动上料超时
ORLD
LDNOT H61.00  ; RK_07 #2铝壳上料升降机构有料记忆
LD H60.00  ; RK_07 #2铝壳上料升降机构手动上料记忆
ANDNOT P_On
ORLD
ANDLD
ANDNOT 817.13  ; RK_07 #2铝壳上料高限位（#3）标志[0017.13]
ANDNOT 2094.13  ; RK_07 U8_Z 铝壳上料移载Y轴忙标志位
AND=(300) D1116 &1  ; RK_07 铝壳上料移载机构步序1（铝壳上料）
AND=(300) D1119 &1  ; RK_07 铝壳上料移载机构步序2（铝壳取料）
AND=(300) D1122 &1  ; RK_07 铝壳上料移载机构步序3（铝壳托盘卸载）
OUT W242.11  ; RK_07 #2铝壳上料电机启动标志
; rung 17: #3铝壳下料电机启动标志
LD 817.01  ; RK_07 #3托盘下料启动按钮标志[0017.01]
AND 814.13  ; RK_07 #3托盘下料车定位升降气缸下降位标志[0014.13]
AND 817.15  ; RK_07 #3托盘下料位物料车到位感应标志[0017.15]
AND 819.14  ; RK_07 #3托盘下料位物料车到位感应#2标志[0019.14]
ANDNOT 117.14  ; RK_07 #3托盘下料电机正转
ANDNOT 117.15  ; RK_07 #3托盘下料电机反转
ANDNOT 817.14  ; RK_07 #3托盘下料上升到位感应标志[0017.14]
ANDNOT 819.13  ; RK_07 #3托盘下料下降到位感应标志[0019.13]
LD W242.12  ; RK_07 #3铝壳下料电机启动标志
AND H65.00  ; RK_07 铝壳托盘下料升降机构手动下料记忆
ANDNOT W80.02  ; #3铝壳托盘下料机构手动下料超时
ORLD
LD H66.00  ; RK_07 铝壳托盘下料升降机构有料记忆
LD H65.00  ; RK_07 铝壳托盘下料升降机构手动下料记忆
ANDNOT P_On
ORLD
ANDLD
OUT W242.12  ; RK_07 #3铝壳下料电机启动标志
; rung 18: #1铝壳上料电机初次上料感应到上料托盘到位信号延时反转启动到安全位
LD W242.10  ; RK_07 #1铝壳上料电机启动标志
AND 817.04  ; RK_07 #1铝壳上料托盘到位感应标志[0017.04]
ANDNOT 117.04  ; RK_07 #1铝壳上料电机正转
ANDNOT 117.05  ; RK_07 #1铝壳上料电机反转
TIMX(550) 2595 &20  ; #1铝壳上料电机初次上料反转到安全位延时
; rung 19: #1铝壳上料电机初次上料延时下降#1铝壳上料车定位升降气缸
LD W242.10  ; RK_07 #1铝壳上料电机启动标志
AND 117.04  ; RK_07 #1铝壳上料电机正转
ANDNOT P_On
TIMX(550) 2596 &50  ; #1铝壳上料车定位升降气缸下降延时

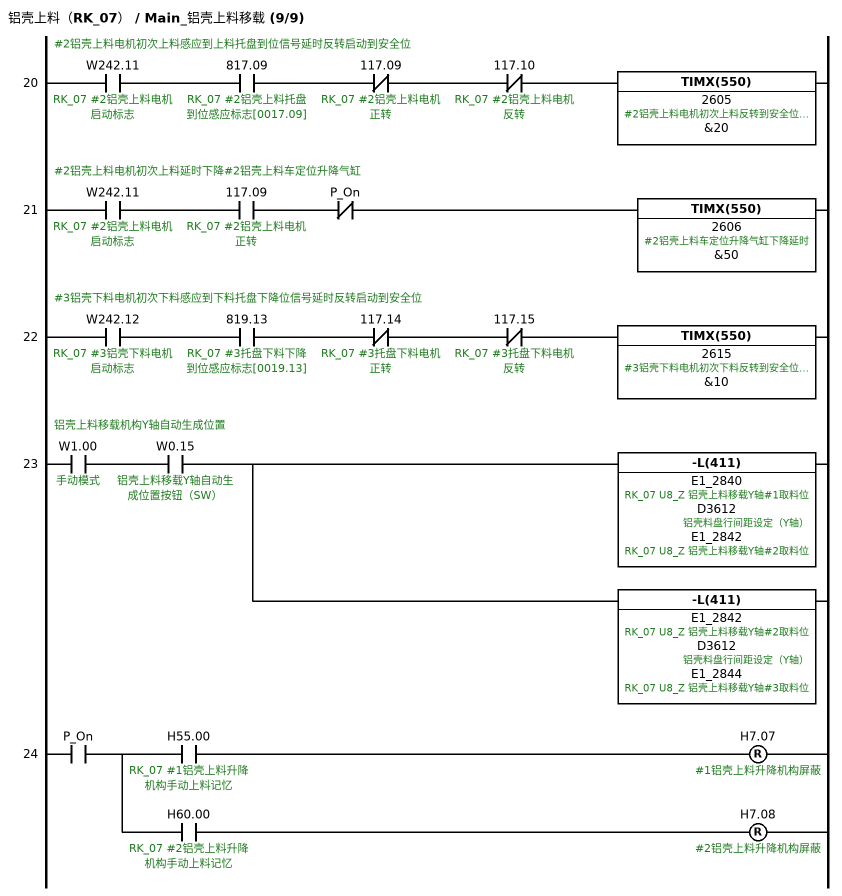
; rung 20: #2铝壳上料电机初次上料感应到上料托盘到位信号延时反转启动到安全位
LD W242.11  ; RK_07 #2铝壳上料电机启动标志
AND 817.09  ; RK_07 #2铝壳上料托盘到位感应标志[0017.09]
ANDNOT 117.09  ; RK_07 #2铝壳上料电机正转
ANDNOT 117.10  ; RK_07 #2铝壳上料电机反转
TIMX(550) 2605 &20  ; #2铝壳上料电机初次上料反转到安全位延时
; rung 21: #2铝壳上料电机初次上料延时下降#2铝壳上料车定位升降气缸
LD W242.11  ; RK_07 #2铝壳上料电机启动标志
AND 117.09  ; RK_07 #2铝壳上料电机正转
ANDNOT P_On
TIMX(550) 2606 &50  ; #2铝壳上料车定位升降气缸下降延时
; rung 22: #3铝壳下料电机初次下料感应到下料托盘下降位信号延时反转启动到安全位
LD W242.12  ; RK_07 #3铝壳下料电机启动标志
AND 819.13  ; RK_07 #3托盘下料下降到位感应标志[0019.13]
ANDNOT 117.14  ; RK_07 #3托盘下料电机正转
ANDNOT 117.15  ; RK_07 #3托盘下料电机反转
TIMX(550) 2615 &10  ; #3铝壳下料电机初次下料反转到安全位延时
; rung 23: 铝壳上料移载机构Y轴自动生成位置
LD W1.00  ; 手动模式
AND W0.15  ; 铝壳上料移载Y轴自动生成位置按钮（SW）
-L(411) E1_2840 D3612 E1_2842  ; RK_07 U8_Z 铝壳上料移载Y轴#1取料位, 铝壳料盘行间距设定（Y轴）, RK_07 U8_Z 铝壳上料移载Y轴#2取料位
-L(411) E1_2842 D3612 E1_2844  ; RK_07 U8_Z 铝壳上料移载Y轴#2取料位, 铝壳料盘行间距设定（Y轴）, RK_07 U8_Z 铝壳上料移载Y轴#3取料位
; rung 24
LD P_On
OUT TR0
AND H55.00  ; RK_07 #1铝壳上料升降机构手动上料记忆
RSET H7.07  ; #1铝壳上料升降机构屏蔽
LD TR0
AND H60.00  ; RK_07 #2铝壳上料升降机构手动上料记忆
RSET H7.08  ; #2铝壳上料升降机构屏蔽

### Section Main_铝壳上下料升降

### Section 手动_铝壳进料

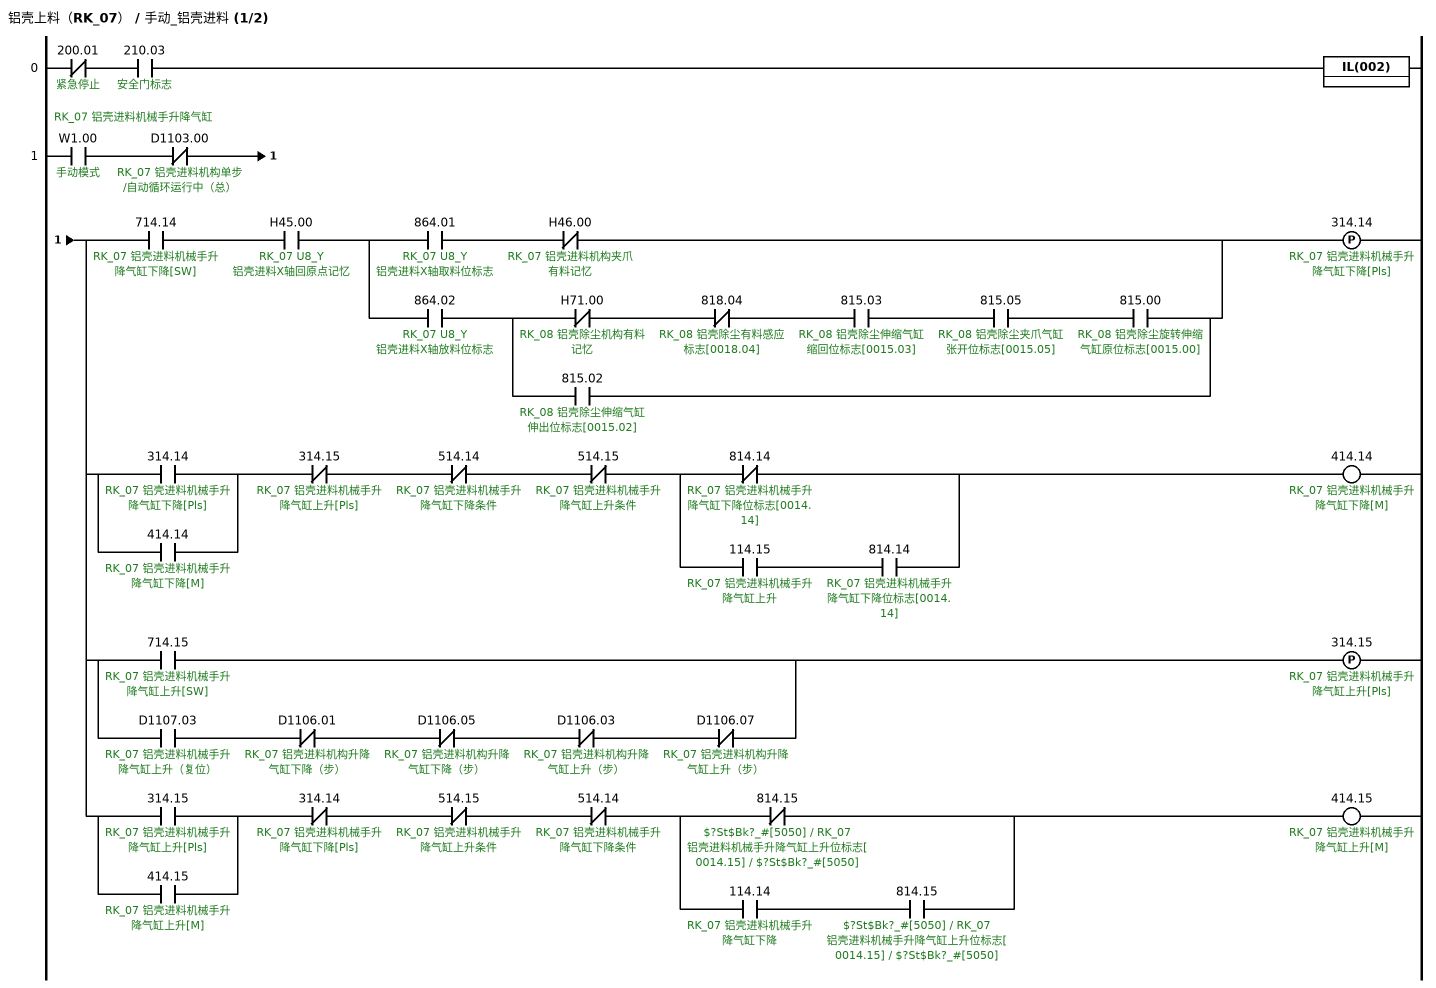
; rung 0
LDNOT 200.01  ; 紧急停止
AND 210.03  ; 安全门标志
IL(002)
; rung 1: RK_07 铝壳进料机械手升降气缸
LD W1.00  ; 手动模式
ANDNOT D1103.00  ; RK_07 铝壳进料机构单步/自动循环运行中（总）
OUT TR0
AND 714.14  ; RK_07 铝壳进料机械手升降气缸下降[SW]
AND H45.00  ; RK_07 U8_Y 铝壳进料X轴回原点记忆
LD 864.01  ; RK_07 U8_Y 铝壳进料X轴取料位标志
ANDNOT H46.00  ; RK_07 铝壳进料机构夹爪有料记忆
LD 864.02  ; RK_07 U8_Y 铝壳进料X轴放料位标志
LDNOT H71.00  ; RK_08 铝壳除尘机构有料记忆
ANDNOT 818.04  ; RK_08 铝壳除尘有料感应标志[0018.04]
AND 815.03  ; RK_08 铝壳除尘伸缩气缸缩回位标志[0015.03]
AND 815.05  ; RK_08 铝壳除尘夹爪气缸张开位标志[0015.05]
AND 815.00  ; RK_08 铝壳除尘旋转伸缩气缸原位标志[0015.00]
OR 815.02  ; RK_08 铝壳除尘伸缩气缸伸出位标志[0015.02]
ANDLD
ORLD
ANDLD
DIFU(013) 314.14  ; RK_07 铝壳进料机械手升降气缸下降[Pls]
LD TR0
LD 314.14  ; RK_07 铝壳进料机械手升降气缸下降[Pls]
OR 414.14  ; RK_07 铝壳进料机械手升降气缸下降[M]
ANDLD
ANDNOT 314.15  ; RK_07 铝壳进料机械手升降气缸上升[Pls]
ANDNOT 514.14  ; RK_07 铝壳进料机械手升降气缸下降条件
ANDNOT 514.15  ; RK_07 铝壳进料机械手升降气缸上升条件
LDNOT 814.14  ; RK_07 铝壳进料机械手升降气缸下降位标志[0014.14]
LD 114.15  ; RK_07 铝壳进料机械手升降气缸上升
AND 814.14  ; RK_07 铝壳进料机械手升降气缸下降位标志[0014.14]
ORLD
ANDLD
OUT 414.14  ; RK_07 铝壳进料机械手升降气缸下降[M]
LD TR0
LD 714.15  ; RK_07 铝壳进料机械手升降气缸上升[SW]
LD D1107.03  ; RK_07 铝壳进料机械手升降气缸上升（复位）
ANDNOT D1106.01  ; RK_07 铝壳进料机构升降气缸下降（步）
ANDNOT D1106.05  ; RK_07 铝壳进料机构升降气缸下降（步）
ANDNOT D1106.03  ; RK_07 铝壳进料机构升降气缸上升（步）
ANDNOT D1106.07  ; RK_07 铝壳进料机构升降气缸上升（步）
ORLD
ANDLD
DIFU(013) 314.15  ; RK_07 铝壳进料机械手升降气缸上升[Pls]
LD TR0
LD 314.15  ; RK_07 铝壳进料机械手升降气缸上升[Pls]
OR 414.15  ; RK_07 铝壳进料机械手升降气缸上升[M]
ANDLD
ANDNOT 314.14  ; RK_07 铝壳进料机械手升降气缸下降[Pls]
ANDNOT 514.15  ; RK_07 铝壳进料机械手升降气缸上升条件
ANDNOT 514.14  ; RK_07 铝壳进料机械手升降气缸下降条件
LDNOT 814.15  ; $?St$Bk?_#[5050] / RK_07 铝壳进料机械手升降气缸上升位标志[0014.15] / $?St$Bk?_#[5050]
LD 114.14  ; RK_07 铝壳进料机械手升降气缸下降
AND 814.15  ; $?St$Bk?_#[5050] / RK_07 铝壳进料机械手升降气缸上升位标志[0014.15] / $?St$Bk?_#[5050]
ORLD
ANDLD
OUT 414.15  ; RK_07 铝壳进料机械手升降气缸上升[M]

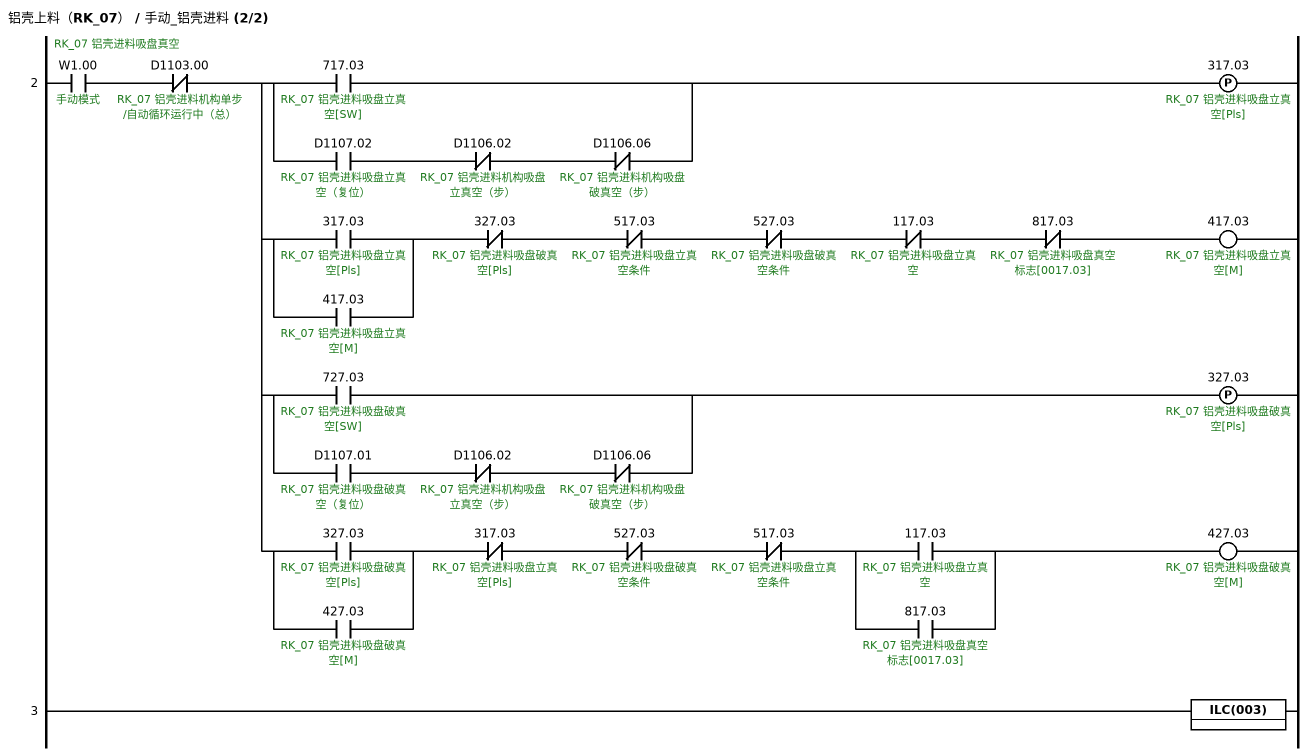
; rung 2: RK_07 铝壳进料吸盘真空
LD W1.00  ; 手动模式
ANDNOT D1103.00  ; RK_07 铝壳进料机构单步/自动循环运行中（总）
OUT TR0
LD 717.03  ; RK_07 铝壳进料吸盘立真空[SW]
LD D1107.02  ; RK_07 铝壳进料吸盘立真空（复位）
ANDNOT D1106.02  ; RK_07 铝壳进料机构吸盘立真空（步）
ANDNOT D1106.06  ; RK_07 铝壳进料机构吸盘破真空（步）
ORLD
ANDLD
DIFU(013) 317.03  ; RK_07 铝壳进料吸盘立真空[Pls]
LD TR0
LD 317.03  ; RK_07 铝壳进料吸盘立真空[Pls]
OR 417.03  ; RK_07 铝壳进料吸盘立真空[M]
ANDLD
ANDNOT 327.03  ; RK_07 铝壳进料吸盘破真空[Pls]
ANDNOT 517.03  ; RK_07 铝壳进料吸盘立真空条件
ANDNOT 527.03  ; RK_07 铝壳进料吸盘破真空条件
ANDNOT 117.03  ; RK_07 铝壳进料吸盘立真空
ANDNOT 817.03  ; RK_07 铝壳进料吸盘真空标志[0017.03]
OUT 417.03  ; RK_07 铝壳进料吸盘立真空[M]
LD TR0
LD 727.03  ; RK_07 铝壳进料吸盘破真空[SW]
LD D1107.01  ; RK_07 铝壳进料吸盘破真空（复位）
ANDNOT D1106.02  ; RK_07 铝壳进料机构吸盘立真空（步）
ANDNOT D1106.06  ; RK_07 铝壳进料机构吸盘破真空（步）
ORLD
ANDLD
DIFU(013) 327.03  ; RK_07 铝壳进料吸盘破真空[Pls]
LD TR0
LD 327.03  ; RK_07 铝壳进料吸盘破真空[Pls]
OR 427.03  ; RK_07 铝壳进料吸盘破真空[M]
ANDLD
ANDNOT 317.03  ; RK_07 铝壳进料吸盘立真空[Pls]
ANDNOT 527.03  ; RK_07 铝壳进料吸盘破真空条件
ANDNOT 517.03  ; RK_07 铝壳进料吸盘立真空条件
LD 117.03  ; RK_07 铝壳进料吸盘立真空
OR 817.03  ; RK_07 铝壳进料吸盘真空标志[0017.03]
ANDLD
OUT 427.03  ; RK_07 铝壳进料吸盘破真空[M]
; rung 3
ILC(003)

### Section 手动_铝壳上料移载

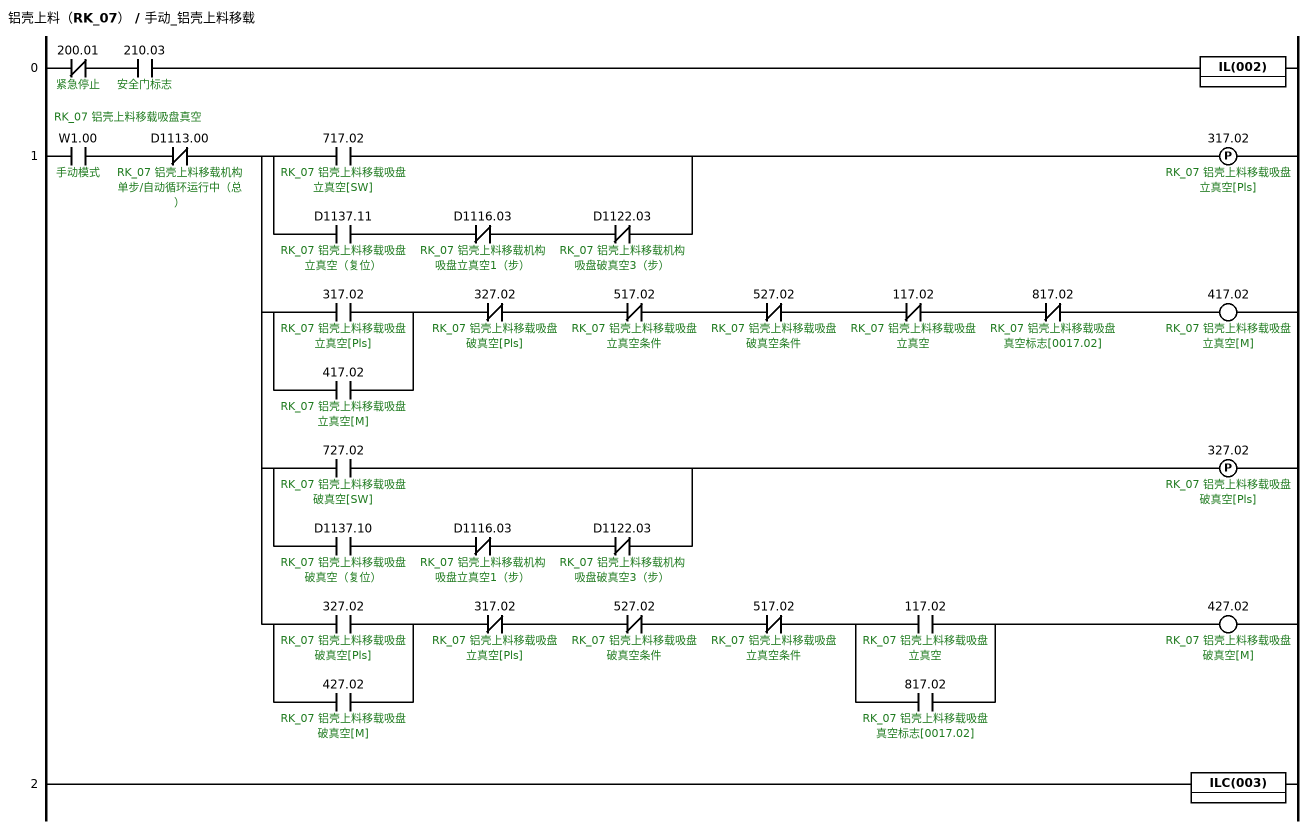
; rung 0
LDNOT 200.01  ; 紧急停止
AND 210.03  ; 安全门标志
IL(002)
; rung 1: RK_07 铝壳上料移载吸盘真空
LD W1.00  ; 手动模式
ANDNOT D1113.00  ; RK_07 铝壳上料移载机构单步/自动循环运行中（总）
OUT TR0
LD 717.02  ; RK_07 铝壳上料移载吸盘立真空[SW]
LD D1137.11  ; RK_07 铝壳上料移载吸盘立真空（复位）
ANDNOT D1116.03  ; RK_07 铝壳上料移载机构吸盘立真空1（步）
ANDNOT D1122.03  ; RK_07 铝壳上料移载机构吸盘破真空3（步）
ORLD
ANDLD
DIFU(013) 317.02  ; RK_07 铝壳上料移载吸盘立真空[Pls]
LD TR0
LD 317.02  ; RK_07 铝壳上料移载吸盘立真空[Pls]
OR 417.02  ; RK_07 铝壳上料移载吸盘立真空[M]
ANDLD
ANDNOT 327.02  ; RK_07 铝壳上料移载吸盘破真空[Pls]
ANDNOT 517.02  ; RK_07 铝壳上料移载吸盘立真空条件
ANDNOT 527.02  ; RK_07 铝壳上料移载吸盘破真空条件
ANDNOT 117.02  ; RK_07 铝壳上料移载吸盘立真空
ANDNOT 817.02  ; RK_07 铝壳上料移载吸盘真空标志[0017.02]
OUT 417.02  ; RK_07 铝壳上料移载吸盘立真空[M]
LD TR0
LD 727.02  ; RK_07 铝壳上料移载吸盘破真空[SW]
LD D1137.10  ; RK_07 铝壳上料移载吸盘破真空（复位）
ANDNOT D1116.03  ; RK_07 铝壳上料移载机构吸盘立真空1（步）
ANDNOT D1122.03  ; RK_07 铝壳上料移载机构吸盘破真空3（步）
ORLD
ANDLD
DIFU(013) 327.02  ; RK_07 铝壳上料移载吸盘破真空[Pls]
LD TR0
LD 327.02  ; RK_07 铝壳上料移载吸盘破真空[Pls]
OR 427.02  ; RK_07 铝壳上料移载吸盘破真空[M]
ANDLD
ANDNOT 317.02  ; RK_07 铝壳上料移载吸盘立真空[Pls]
ANDNOT 527.02  ; RK_07 铝壳上料移载吸盘破真空条件
ANDNOT 517.02  ; RK_07 铝壳上料移载吸盘立真空条件
LD 117.02  ; RK_07 铝壳上料移载吸盘立真空
OR 817.02  ; RK_07 铝壳上料移载吸盘真空标志[0017.02]
ANDLD
OUT 427.02  ; RK_07 铝壳上料移载吸盘破真空[M]
; rung 2
ILC(003)

### Section 手动_铝壳上下料升降

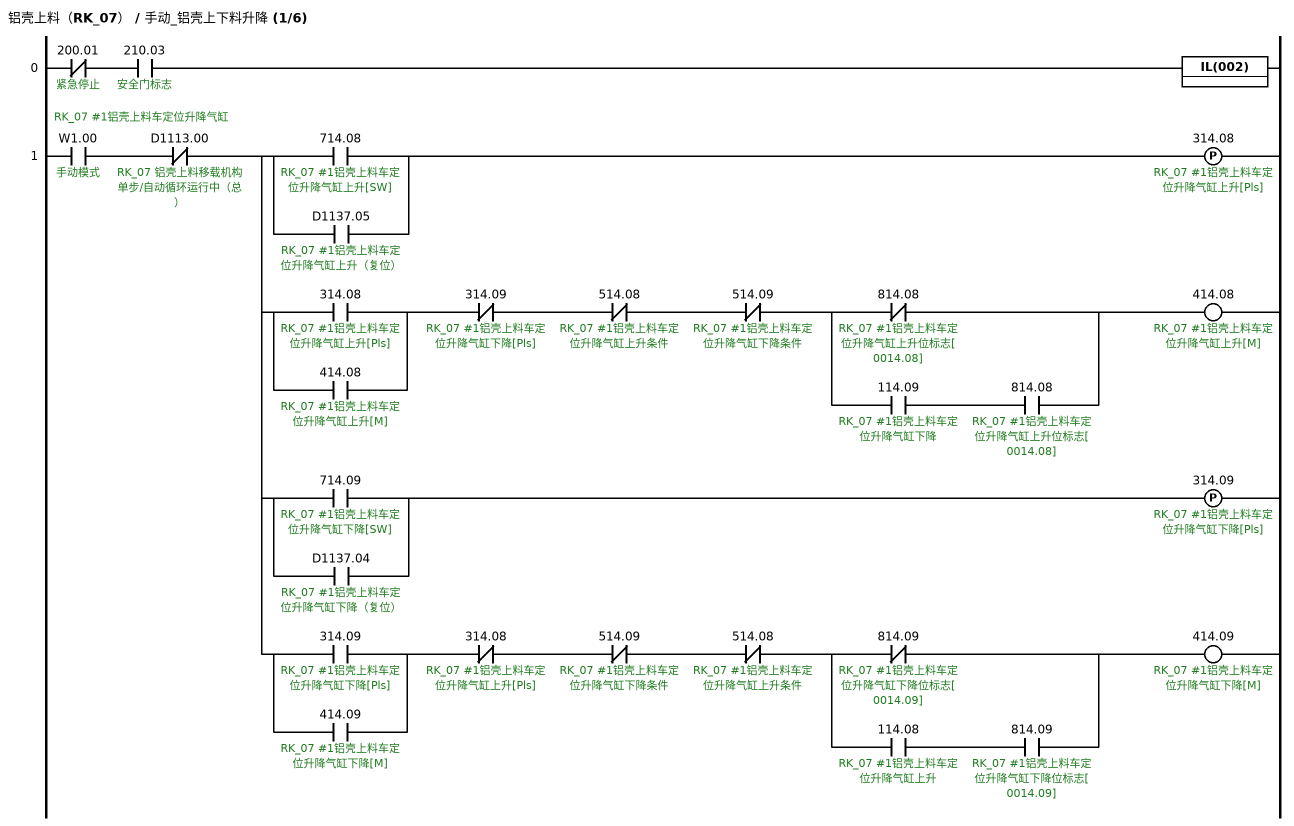
; rung 0
LDNOT 200.01  ; 紧急停止
AND 210.03  ; 安全门标志
IL(002)
; rung 1: RK_07 #1铝壳上料车定位升降气缸
LD W1.00  ; 手动模式
ANDNOT D1113.00  ; RK_07 铝壳上料移载机构单步/自动循环运行中（总）
OUT TR0
LD 714.08  ; RK_07 #1铝壳上料车定位升降气缸上升[SW]
OR D1137.05  ; RK_07 #1铝壳上料车定位升降气缸上升（复位）
ANDLD
DIFU(013) 314.08  ; RK_07 #1铝壳上料车定位升降气缸上升[Pls]
LD TR0
LD 314.08  ; RK_07 #1铝壳上料车定位升降气缸上升[Pls]
OR 414.08  ; RK_07 #1铝壳上料车定位升降气缸上升[M]
ANDLD
ANDNOT 314.09  ; RK_07 #1铝壳上料车定位升降气缸下降[Pls]
ANDNOT 514.08  ; RK_07 #1铝壳上料车定位升降气缸上升条件
ANDNOT 514.09  ; RK_07 #1铝壳上料车定位升降气缸下降条件
LDNOT 814.08  ; RK_07 #1铝壳上料车定位升降气缸上升位标志[0014.08]
LD 114.09  ; RK_07 #1铝壳上料车定位升降气缸下降
AND 814.08  ; RK_07 #1铝壳上料车定位升降气缸上升位标志[0014.08]
ORLD
ANDLD
OUT 414.08  ; RK_07 #1铝壳上料车定位升降气缸上升[M]
LD TR0
LD 714.09  ; RK_07 #1铝壳上料车定位升降气缸下降[SW]
OR D1137.04  ; RK_07 #1铝壳上料车定位升降气缸下降（复位）
ANDLD
DIFU(013) 314.09  ; RK_07 #1铝壳上料车定位升降气缸下降[Pls]
LD TR0
LD 314.09  ; RK_07 #1铝壳上料车定位升降气缸下降[Pls]
OR 414.09  ; RK_07 #1铝壳上料车定位升降气缸下降[M]
ANDLD
ANDNOT 314.08  ; RK_07 #1铝壳上料车定位升降气缸上升[Pls]
ANDNOT 514.09  ; RK_07 #1铝壳上料车定位升降气缸下降条件
ANDNOT 514.08  ; RK_07 #1铝壳上料车定位升降气缸上升条件
LDNOT 814.09  ; RK_07 #1铝壳上料车定位升降气缸下降位标志[0014.09]
LD 114.08  ; RK_07 #1铝壳上料车定位升降气缸上升
AND 814.09  ; RK_07 #1铝壳上料车定位升降气缸下降位标志[0014.09]
ORLD
ANDLD
OUT 414.09  ; RK_07 #1铝壳上料车定位升降气缸下降[M]

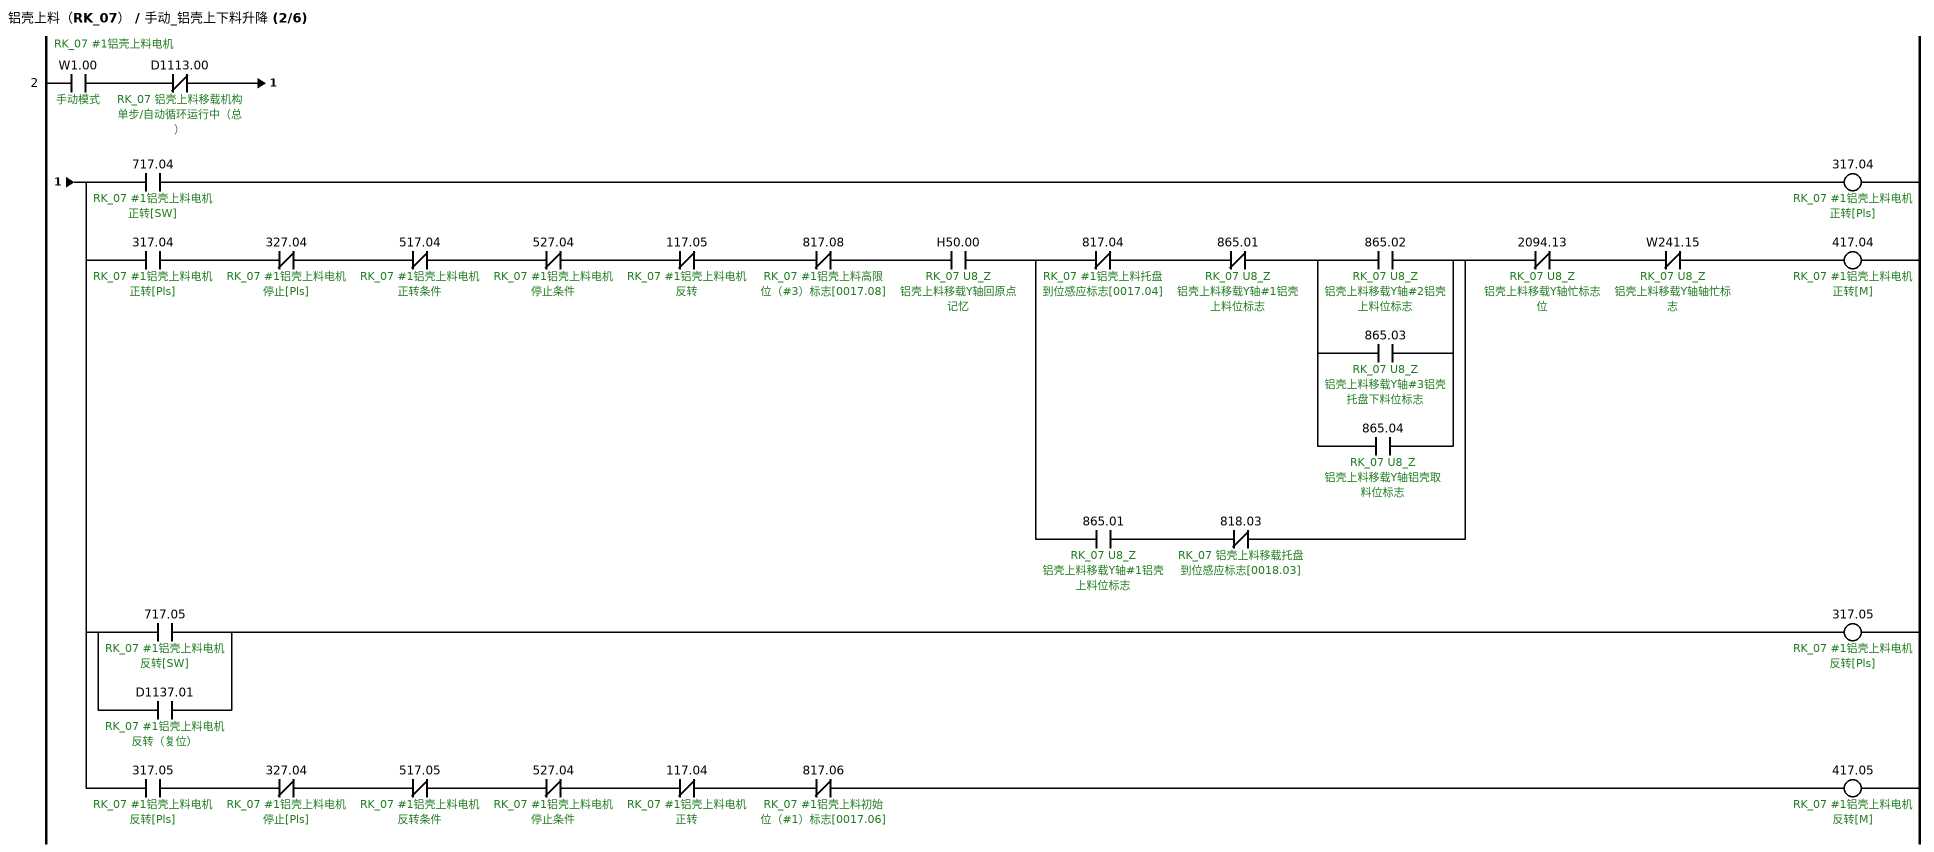
; rung 2: RK_07 #1铝壳上料电机
LD W1.00  ; 手动模式
ANDNOT D1113.00  ; RK_07 铝壳上料移载机构单步/自动循环运行中（总）
OUT TR0
AND 717.04  ; RK_07 #1铝壳上料电机正转[SW]
OUT 317.04  ; RK_07 #1铝壳上料电机正转[Pls]
LD TR0
AND 317.04  ; RK_07 #1铝壳上料电机正转[Pls]
ANDNOT 327.04  ; RK_07 #1铝壳上料电机停止[Pls]
ANDNOT 517.04  ; RK_07 #1铝壳上料电机正转条件
ANDNOT 527.04  ; RK_07 #1铝壳上料电机停止条件
ANDNOT 117.05  ; RK_07 #1铝壳上料电机反转
ANDNOT 817.08  ; RK_07 #1铝壳上料高限位（#3）标志[0017.08]
AND H50.00  ; RK_07 U8_Z 铝壳上料移载Y轴回原点记忆
LDNOT 817.04  ; RK_07 #1铝壳上料托盘到位感应标志[0017.04]  // 手动模式加此联锁！
ANDNOT 865.01  ; RK_07 U8_Z 铝壳上料移载Y轴#1铝壳上料位标志
LD 865.02  ; RK_07 U8_Z 铝壳上料移载Y轴#2铝壳上料位标志
OR 865.03  ; RK_07 U8_Z 铝壳上料移载Y轴#3铝壳托盘下料位标志
OR 865.04  ; RK_07 U8_Z 铝壳上料移载Y轴铝壳取料位标志
ANDLD
LD 865.01  ; RK_07 U8_Z 铝壳上料移载Y轴#1铝壳上料位标志
ANDNOT 818.03  ; RK_07 铝壳上料移载托盘到位感应标志[0018.03]
ORLD
ANDLD
ANDNOT 2094.13  ; RK_07 U8_Z 铝壳上料移载Y轴忙标志位
ANDNOT W241.15  ; RK_07 U8_Z 铝壳上料移载Y轴轴忙标志
OUT 417.04  ; RK_07 #1铝壳上料电机正转[M]
LD TR0
LD 717.05  ; RK_07 #1铝壳上料电机反转[SW]
OR D1137.01  ; RK_07 #1铝壳上料电机反转（复位）
ANDLD
OUT 317.05  ; RK_07 #1铝壳上料电机反转[Pls]
LD TR0
AND 317.05  ; RK_07 #1铝壳上料电机反转[Pls]
ANDNOT 327.04  ; RK_07 #1铝壳上料电机停止[Pls]
ANDNOT 517.05  ; RK_07 #1铝壳上料电机反转条件
ANDNOT 527.04  ; RK_07 #1铝壳上料电机停止条件
ANDNOT 117.04  ; RK_07 #1铝壳上料电机正转
ANDNOT 817.06  ; RK_07 #1铝壳上料初始位（#1）标志[0017.06]
OUT 417.05  ; RK_07 #1铝壳上料电机反转[M]

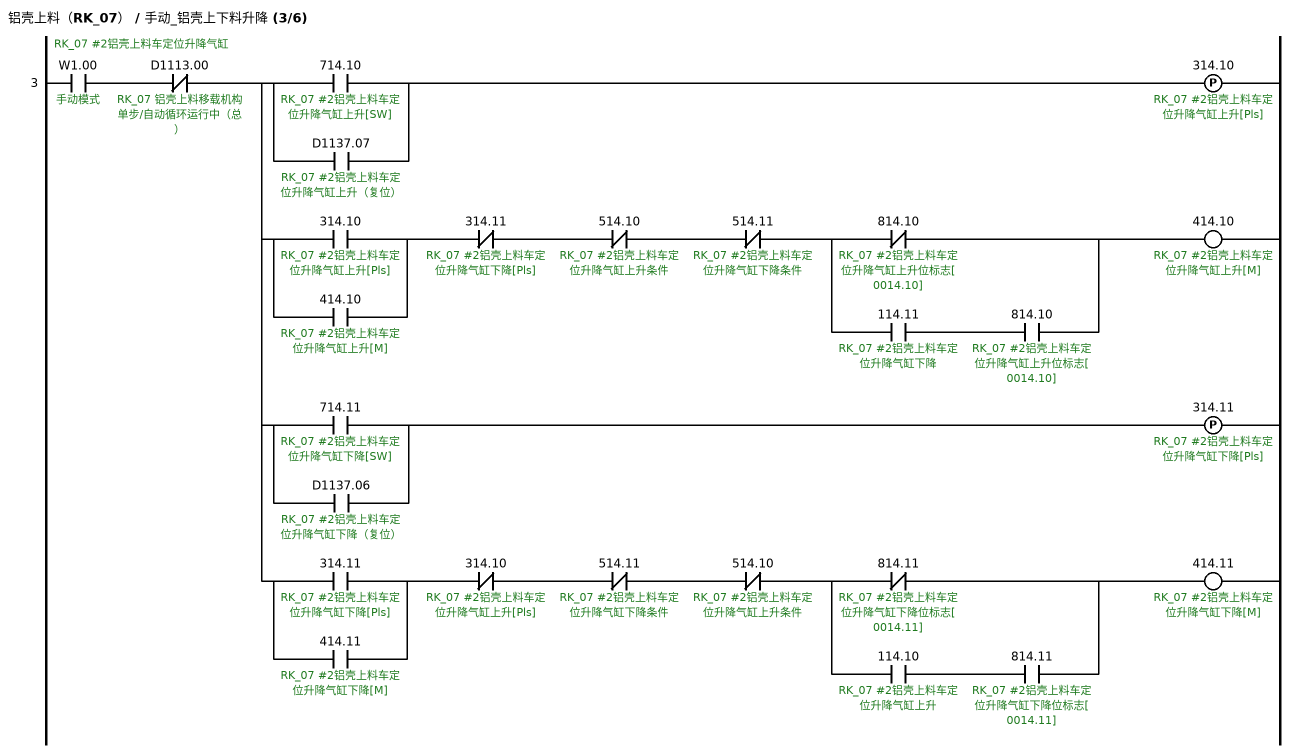
; rung 3: RK_07 #2铝壳上料车定位升降气缸
LD W1.00  ; 手动模式
ANDNOT D1113.00  ; RK_07 铝壳上料移载机构单步/自动循环运行中（总）
OUT TR0
LD 714.10  ; RK_07 #2铝壳上料车定位升降气缸上升[SW]
OR D1137.07  ; RK_07 #2铝壳上料车定位升降气缸上升（复位）
ANDLD
DIFU(013) 314.10  ; RK_07 #2铝壳上料车定位升降气缸上升[Pls]
LD TR0
LD 314.10  ; RK_07 #2铝壳上料车定位升降气缸上升[Pls]
OR 414.10  ; RK_07 #2铝壳上料车定位升降气缸上升[M]
ANDLD
ANDNOT 314.11  ; RK_07 #2铝壳上料车定位升降气缸下降[Pls]
ANDNOT 514.10  ; RK_07 #2铝壳上料车定位升降气缸上升条件
ANDNOT 514.11  ; RK_07 #2铝壳上料车定位升降气缸下降条件
LDNOT 814.10  ; RK_07 #2铝壳上料车定位升降气缸上升位标志[0014.10]
LD 114.11  ; RK_07 #2铝壳上料车定位升降气缸下降
AND 814.10  ; RK_07 #2铝壳上料车定位升降气缸上升位标志[0014.10]
ORLD
ANDLD
OUT 414.10  ; RK_07 #2铝壳上料车定位升降气缸上升[M]
LD TR0
LD 714.11  ; RK_07 #2铝壳上料车定位升降气缸下降[SW]
OR D1137.06  ; RK_07 #2铝壳上料车定位升降气缸下降（复位）
ANDLD
DIFU(013) 314.11  ; RK_07 #2铝壳上料车定位升降气缸下降[Pls]
LD TR0
LD 314.11  ; RK_07 #2铝壳上料车定位升降气缸下降[Pls]
OR 414.11  ; RK_07 #2铝壳上料车定位升降气缸下降[M]
ANDLD
ANDNOT 314.10  ; RK_07 #2铝壳上料车定位升降气缸上升[Pls]
ANDNOT 514.11  ; RK_07 #2铝壳上料车定位升降气缸下降条件
ANDNOT 514.10  ; RK_07 #2铝壳上料车定位升降气缸上升条件
LDNOT 814.11  ; RK_07 #2铝壳上料车定位升降气缸下降位标志[0014.11]
LD 114.10  ; RK_07 #2铝壳上料车定位升降气缸上升
AND 814.11  ; RK_07 #2铝壳上料车定位升降气缸下降位标志[0014.11]
ORLD
ANDLD
OUT 414.11  ; RK_07 #2铝壳上料车定位升降气缸下降[M]

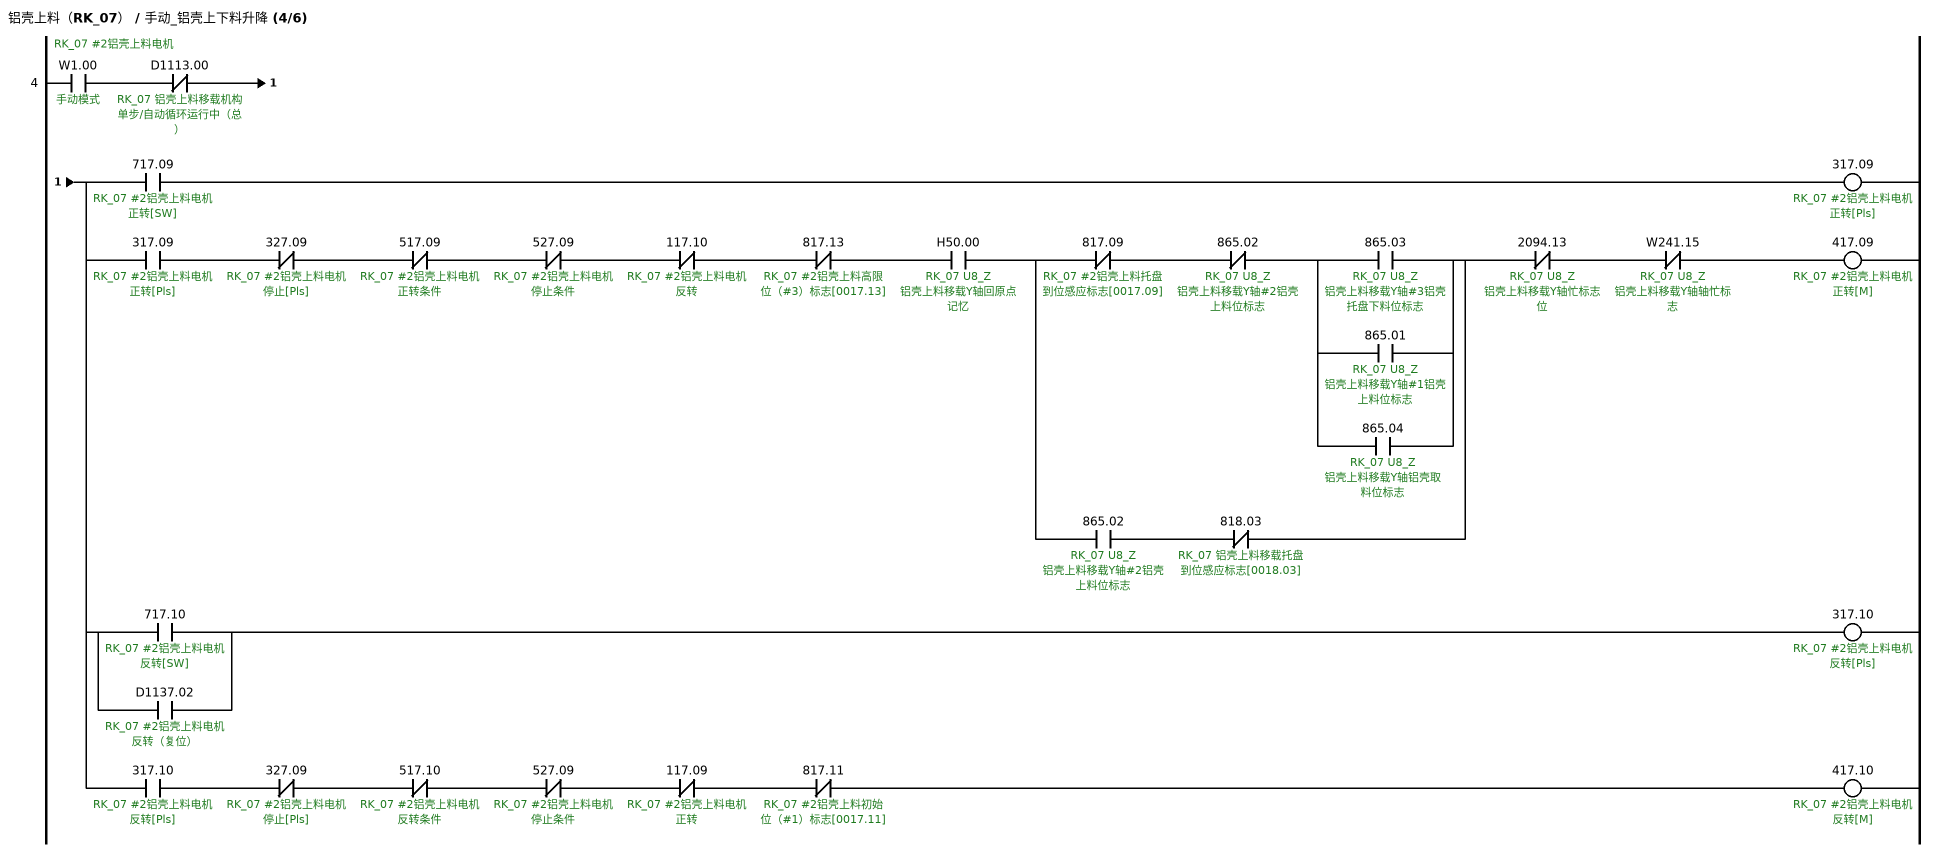
; rung 4: RK_07 #2铝壳上料电机
LD W1.00  ; 手动模式
ANDNOT D1113.00  ; RK_07 铝壳上料移载机构单步/自动循环运行中（总）
OUT TR0
AND 717.09  ; RK_07 #2铝壳上料电机正转[SW]
OUT 317.09  ; RK_07 #2铝壳上料电机正转[Pls]
LD TR0
AND 317.09  ; RK_07 #2铝壳上料电机正转[Pls]
ANDNOT 327.09  ; RK_07 #2铝壳上料电机停止[Pls]
ANDNOT 517.09  ; RK_07 #2铝壳上料电机正转条件
ANDNOT 527.09  ; RK_07 #2铝壳上料电机停止条件
ANDNOT 117.10  ; RK_07 #2铝壳上料电机反转
ANDNOT 817.13  ; RK_07 #2铝壳上料高限位（#3）标志[0017.13]
AND H50.00  ; RK_07 U8_Z 铝壳上料移载Y轴回原点记忆
LDNOT 817.09  ; RK_07 #2铝壳上料托盘到位感应标志[0017.09]  // 手动模式加此联锁！
ANDNOT 865.02  ; RK_07 U8_Z 铝壳上料移载Y轴#2铝壳上料位标志
LD 865.03  ; RK_07 U8_Z 铝壳上料移载Y轴#3铝壳托盘下料位标志
OR 865.01  ; RK_07 U8_Z 铝壳上料移载Y轴#1铝壳上料位标志
OR 865.04  ; RK_07 U8_Z 铝壳上料移载Y轴铝壳取料位标志
ANDLD
LD 865.02  ; RK_07 U8_Z 铝壳上料移载Y轴#2铝壳上料位标志
ANDNOT 818.03  ; RK_07 铝壳上料移载托盘到位感应标志[0018.03]
ORLD
ANDLD
ANDNOT 2094.13  ; RK_07 U8_Z 铝壳上料移载Y轴忙标志位
ANDNOT W241.15  ; RK_07 U8_Z 铝壳上料移载Y轴轴忙标志
OUT 417.09  ; RK_07 #2铝壳上料电机正转[M]
LD TR0
LD 717.10  ; RK_07 #2铝壳上料电机反转[SW]
OR D1137.02  ; RK_07 #2铝壳上料电机反转（复位）
ANDLD
OUT 317.10  ; RK_07 #2铝壳上料电机反转[Pls]
LD TR0
AND 317.10  ; RK_07 #2铝壳上料电机反转[Pls]
ANDNOT 327.09  ; RK_07 #2铝壳上料电机停止[Pls]
ANDNOT 517.10  ; RK_07 #2铝壳上料电机反转条件
ANDNOT 527.09  ; RK_07 #2铝壳上料电机停止条件
ANDNOT 117.09  ; RK_07 #2铝壳上料电机正转
ANDNOT 817.11  ; RK_07 #2铝壳上料初始位（#1）标志[0017.11]
OUT 417.10  ; RK_07 #2铝壳上料电机反转[M]

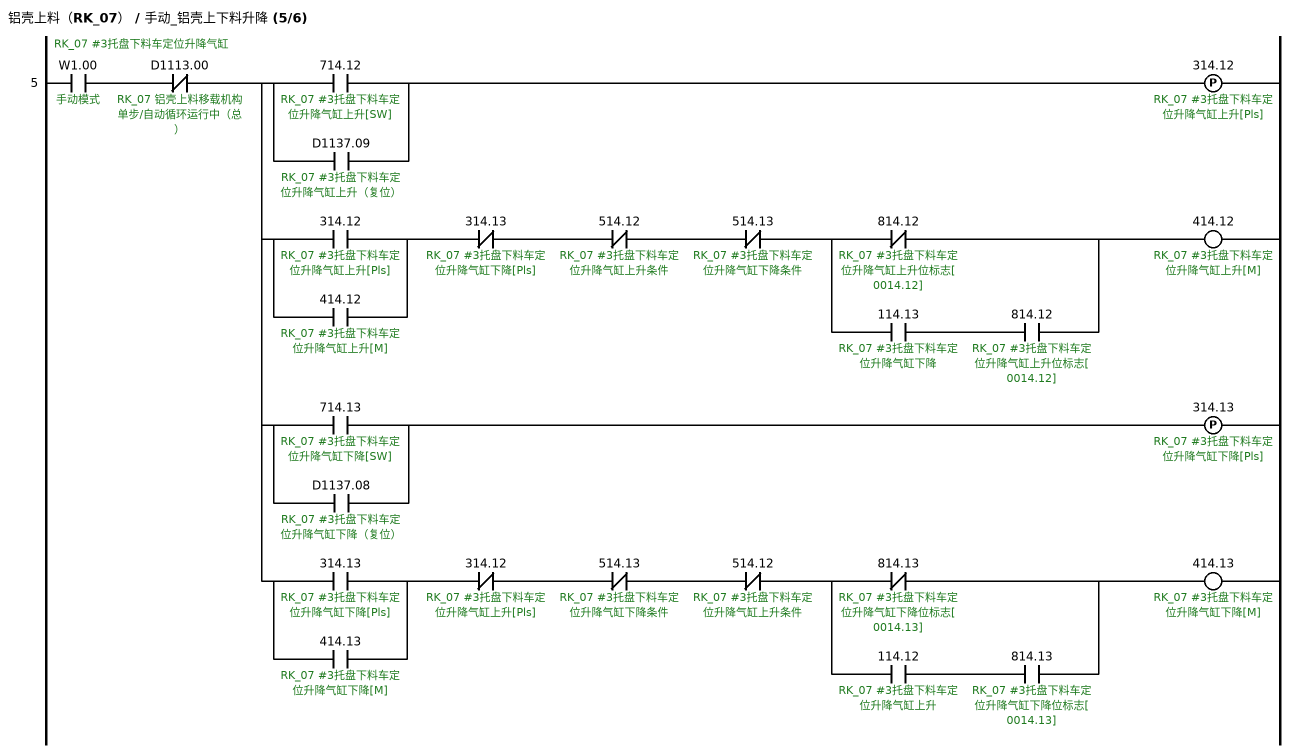
; rung 5: RK_07 #3托盘下料车定位升降气缸
LD W1.00  ; 手动模式
ANDNOT D1113.00  ; RK_07 铝壳上料移载机构单步/自动循环运行中（总）
OUT TR0
LD 714.12  ; RK_07 #3托盘下料车定位升降气缸上升[SW]
OR D1137.09  ; RK_07 #3托盘下料车定位升降气缸上升（复位）
ANDLD
DIFU(013) 314.12  ; RK_07 #3托盘下料车定位升降气缸上升[Pls]
LD TR0
LD 314.12  ; RK_07 #3托盘下料车定位升降气缸上升[Pls]
OR 414.12  ; RK_07 #3托盘下料车定位升降气缸上升[M]
ANDLD
ANDNOT 314.13  ; RK_07 #3托盘下料车定位升降气缸下降[Pls]
ANDNOT 514.12  ; RK_07 #3托盘下料车定位升降气缸上升条件
ANDNOT 514.13  ; RK_07 #3托盘下料车定位升降气缸下降条件
LDNOT 814.12  ; RK_07 #3托盘下料车定位升降气缸上升位标志[0014.12]
LD 114.13  ; RK_07 #3托盘下料车定位升降气缸下降
AND 814.12  ; RK_07 #3托盘下料车定位升降气缸上升位标志[0014.12]
ORLD
ANDLD
OUT 414.12  ; RK_07 #3托盘下料车定位升降气缸上升[M]
LD TR0
LD 714.13  ; RK_07 #3托盘下料车定位升降气缸下降[SW]
OR D1137.08  ; RK_07 #3托盘下料车定位升降气缸下降（复位）
ANDLD
DIFU(013) 314.13  ; RK_07 #3托盘下料车定位升降气缸下降[Pls]
LD TR0
LD 314.13  ; RK_07 #3托盘下料车定位升降气缸下降[Pls]
OR 414.13  ; RK_07 #3托盘下料车定位升降气缸下降[M]
ANDLD
ANDNOT 314.12  ; RK_07 #3托盘下料车定位升降气缸上升[Pls]
ANDNOT 514.13  ; RK_07 #3托盘下料车定位升降气缸下降条件
ANDNOT 514.12  ; RK_07 #3托盘下料车定位升降气缸上升条件
LDNOT 814.13  ; RK_07 #3托盘下料车定位升降气缸下降位标志[0014.13]
LD 114.12  ; RK_07 #3托盘下料车定位升降气缸上升
AND 814.13  ; RK_07 #3托盘下料车定位升降气缸下降位标志[0014.13]
ORLD
ANDLD
OUT 414.13  ; RK_07 #3托盘下料车定位升降气缸下降[M]

